(* CoDeSys 2.3 project: cy-221-wg-002.pro *)
(* Title: ClevergyAS - Albino E-02 *)
(* Version: 1.25 *)
(* Author: Andrea Ravasio *)
(* Libraries: mod_com.lib 2.12.10 13:48:32, SerComm.lib 31.5.11 07:54:36, Serial_Interface_01.lib 22.4.13 11:50:14, Standard.lib 2.12.10 13:48:34, SysLibTime.lib 2.12.10 13:48:32, Util.lib 26.9.14 09:12:46, Modb_l05.lib 13.5.15 09:30:08, Visual.lib 2.12.10 13:48:34, Ethernet.lib 2.12.10 13:48:32, WagoLibIdent.lib 25.2.13 10:12:16, WagoLibMBX_01.lib 20.3.12 15:32:40, WagoLibStatus.lib 2.12.10 13:48:32, SysLibFile.lib 2.12.10 13:48:34, SysLibRtc.lib 2.12.10 13:48:32, SysLibSockets.lib 10.2.11 08:20:54, SysLibEvent.lib 2.12.10 13:48:34, SysLibPlcCtrl.lib 2.12.10 13:48:32, SysLibCallback.lib 2.12.10 13:48:32, WagoLibModbus_IP_01.lib 24.7.13 14:05:58, WagoLibInfo.lib 25.2.13 09:58:44 *)

(* PLC configuration (modules and I/O channels)
0750-0402 4 DI 24 V DC 3.0ms [Type_1_4_Channels] node 0, in %IB0 out %QB0 {INTTypePAAssignment = PLC; INTTypeModule = plugged}
  AT %IX0.0 [BOOLOnX_I] Ch_1 Digital input
  AT %IX0.1 [BOOLOnX_I] Ch_2 Digital input
  AT %IX0.2 [BOOLOnX_I] Ch_3 Digital input
  AT %IX0.3 [BOOLOnX_I] Ch_4 Digital input
Fieldbus variables [FB_VARS] node 1, in %IB0 out %QB0
Flag variables [FLAG_VARS] node 2, in %IB0 out %QB0
Modbus-Master [MB_MASTER] node 3, in %IB0 out %QB0
*)

(* Global variable list: Addiitonal_Constants *)
VAR_GLOBAL CONSTANT

	Logger_MaxBCK : WORD:=100;

END_VAR

(* Global variable list: Additional_Retain *)
VAR_GLOBAL RETAIN PERSISTENT
	LogBCKIndex:  WORD;
END_VAR

(* Global variable list: Global_Constants *)
VAR_GLOBAL CONSTANT

	Plant_NAME		: STRING :='cySN:221  cyVER:0 - EGM Impianto Luci ';
	Plant_SN			: DWORD  :=221; 	         (* S/N Impianto di telecontrollo *)
	Plant_SW_VER		: WORD   :=0;		(* Versione SW installata *)


	(* Plant-dependent constants *)
	MAX_LUXNUM 								: INT :=12;
	MAX_LuxElement							: INT :=12;

	(* Filesystem *)
	FilesPath  			: STRING :='S:\';

	(* TCP Logger *)
	Logger_SERVER		: STRING:='';
	Logger_IP			: STRING:='178.33.227.41'; (*'192.168.100.3';*)
	Logger_PORT			: WORD  :=80;
	Logger_GETSTART		: STRING:='GET /cygmsrv/hsgm.ashx?';
	Logger_GETEND		: STRING:='$R$N$R$N';
	Logger_CHECK		: STRING:='True';
	Logger_CRLF			: STRING:='$R$N';
	Logger_DataFile		: STRING:='S:\LOG.DAT';
	Logger_DataFileOld	: STRING:='S:\LOG.BCK';
	Logger_IndexFile	: STRING:='S:\LOG.IDX';
	Logger_ConnRetries	: BYTE:=5;
	Logger_RecoverMsgs	: BYTE:=25;

	(* TCP Remote *)
	Remote_PORT			: WORD  :=10;
	Remote_WELCOME		: STRING:='Connected$R$N';
	Remote_OK			: STRING:='OK$R$N';
	Remote_ERROR		: STRING:='ERROR$R$N';

	(* TCP Sockets *)
	MAX_SEND_TCP_SERVER					 : DWORD:=60000;(*60000*)
	MAX_RECEIVE_TCP_SERVER				 : DWORD:=3000;
	MAX_RECEIVE_TCP_SERVER_SOCKET	 	 : DWORD:=3000;
	MAX_SEND_TCP_CLIENT					 : DWORD:=21000;(*15000*)
	MAX_RECEIVE_TCP_CLIENT				 : DWORD:=3000;
	MAX_RECEIVE_TCP_CLIENT_SOCKET		 : DWORD:=3000;
	MAX_RECEIVE_UDP_SERVER				 : INT  :=1472;
	MAX_RECEIVE_UDP_CLIENT				 : INT  :=1472;
	CONNECT_WATCHDOG_TIME				 : TIME :=t#10s;


	(* VISU COLORS *)
	COLOR_RED 			: DWORD:=16#2020F0;
	COLOR_YELLOW		: DWORD:=16#20F0F0;
	COLOR_GREEN			: DWORD:=16#20F020;
	COLOR_GREEN_OFF 	: DWORD:=16#006000;
	COLOR_LBLUE			: DWORD:=16#F0F080;
	COLOR_LIGHT_GREEN	: DWORD := 16#006000;


END_VAR

(* Global variable list: Global_Retain *)
VAR_GLOBAL RETAIN PERSISTENT

	Mode_Manual : BOOL := FALSE;

	WORKINGTIME_n : ARRAY[1..MAX_LUXNUM] OF DWORD;
	POWERONCYCLES_n : ARRAY[1..MAX_LUXNUM] OF WORD;
	ENERGYCOUNTER_n  : ARRAY[1..MAX_LUXNUM] OF WORD;
	ENERGYCOUNTER_T_n : ARRAY[1..MAX_LUXNUM] OF DWORD;

END_VAR

(* Global variable list: Global_Variables *)
VAR_GLOBAL

	SYS    : typ_SYS;
	Logger : typ_Logger;

	Lamp	:	LAMP_AL_GENERALE;
	LAMP_AL:BOOL; (* Dichiarata perchè non c'è l'uscita fisica *)
	T_AMB	:	INT;		(* Environment temperature *)

	(* Nodi Ethernet *)

	(* Analizzatori di rete Lovato DME 310 T2 *)
	ANZ01	:obj_Anz_Lovato_ETH := (ID:=1, IP:='192.168.2.84');		(* FONDERIA - CONTATORE N.1 *)
	ANZ02	:obj_Anz_Lovato_ETH := (ID:=2, IP:='192.168.2.85');		(* FONDERIA - CONTATORE N.2 *)
	ANZ03	:obj_Anz_Lovato_ETH := (ID:=3, IP:='192.168.2.86');		(* CAMPATA 1-2 - CONTATORE N.3*)
	ANZ04	:obj_Anz_Lovato_ETH := (ID:=4, IP:='192.168.2.87');		(* CAMPATA 3 - CONTATORE N.4 *)
	ANZ05	:obj_Anz_Lovato_ETH := (ID:=5, IP:='192.168.2.88');		(* CAMPATA 4 - CONTATORE N.5 *)
	ANZ06	:obj_Anz_Lovato_ETH := (ID:=6, IP:='192.168.2.89');		(* CAMPATA 5 - CONTATORE N.6 *)
	ANZ07	:obj_Anz_Lovato_ETH := (ID:=7, IP:='192.168.2.90');		(* CAMPATA 6 - CONTATORE N.7 *)
	ANZ08	:obj_Anz_Lovato_ETH := (ID:=8, IP:='192.168.2.91');		(* CAMPATA 7 - CONTATORE N.8 *)
	ANZ09	:obj_Anz_Lovato_ETH := (ID:=9, IP:='192.168.2.92');		(* CAMPATA 8 - CONTATORE N.9 *)
	ANZ10	:obj_Anz_Lovato_ETH := (ID:=10, IP:='192.168.2.93');		(* CAMPATA 9 - CONTATORE N.10 *)
	ANZ11	:obj_Anz_Lovato_ETH := (ID:=11, IP:='192.168.2.94');		(* MAGAZZINO - CONTATORE N.11 *)


	(* Nodi di rete I/ remoto SENECA ZE-4DI-2AI-2DO *)
	NODO01	:obj_Anz_Seneca_ETH := (ID:=1, IP:='192.168.2.95');		(* FONDERIA - CONTATORE N.1 e FONDERIA - CONTATORE N.2*)
	NODO02	:obj_Anz_Seneca_ETH := (ID:=2, IP:='192.168.2.96');		(* CAMPATA 1-2 - CONTATORE N.3 *)
	NODO03	:obj_Anz_Seneca_ETH := (ID:=3, IP:='192.168.2.97');		(* CAMPATA 3 - CONTATORE N.4 *)
	NODO04	:obj_Anz_Seneca_ETH := (ID:=4, IP:='192.168.2.98');		(* CAMPATA 4 - CONTATORE N.5 *)
	NODO05	:obj_Anz_Seneca_ETH := (ID:=5, IP:='192.168.2.99');		(* CAMPATA 5 - CONTATORE N.6 *)
	NODO06	:obj_Anz_Seneca_ETH := (ID:=6, IP:='192.168.2.103');		(* CAMPATA 6 - CONTATORE N.7 *)
	NODO07	:obj_Anz_Seneca_ETH := (ID:=7, IP:='192.168.2.104');		(* CAMPATA 7 - CONTATORE N.8 *)
	NODO08	:obj_Anz_Seneca_ETH := (ID:=8, IP:='192.168.2.105');		(* CAMPATA 8 - CONTATORE N.9 *)
	NODO09	:obj_Anz_Seneca_ETH := (ID:=9, IP:='192.168.2.107');		(* CAMPATA 9 - CONTATORE N.10 *)
	NODO10	:obj_Anz_Seneca_ETH := (ID:=10, IP:='192.168.2.106');	(* MAGAZZINO - CONTATORE N.11 *)

(*	LuxElement : ARRAY[1..MAX_LuxElement] OF obj_LUX:=( dimmingtype:=0, CTRL_MODE:=2,CTRL_MODE_BackUp:=2, KeyQty:=1, KeyMode:=SWITCH_NO);
	TabDefaultLux : ARRAY[1..MAX_LuxElement] OF type_TabListLux :=(LuxNumber:=1, Mode:=2) ; *)
 
	LuxElement01: 	obj_LuxSimple:=( ID:=1,CTRL_MODE:=2);
	LuxElement02: 	obj_LuxSimple:=( ID:=2,CTRL_MODE:=2);
	LuxElement03: 	obj_LuxSimple:=( ID:=3, CTRL_MODE:=2);
	LuxElement04: 	obj_LuxSimple:=( ID:=4, CTRL_MODE:=2);
	LuxElement05: 	obj_LuxSimple:=( ID:=5, CTRL_MODE:=2);
	LuxElement06: 	obj_LuxSimple:=( ID:=6, CTRL_MODE:=2);
	LuxElement07: 	obj_LuxSimple:=( ID:=7, CTRL_MODE:=2);
	LuxElement08: 	obj_LuxSimple:=( ID:=8, CTRL_MODE:=2);
	LuxElement09: 	obj_LuxSimple:=( ID:=9, CTRL_MODE:=2);
	LuxElement10: 	obj_LuxSimple:=( ID:=10, CTRL_MODE:=2);
	LuxElement11: 	obj_LuxSimple:=( ID:=11, CTRL_MODE:=2);
	LuxElement12: 	obj_LuxSimple:=( ID:=12, CTRL_MODE:=2);


	(* Crono per gestione accensioni luci impostazione lux *)
	CRON01	:	obj_CRONTER_01 := (ID:=1, Local_MaxRunTAmb:=5000,Histeresys:=50,TipoCrono:='CRONG'(* Riferimento nle file LOG *));
	CRON02	:	obj_CRONTER_01 := (ID:=2, Local_MaxRunTAmb:=5000,Histeresys:=50,TipoCrono:='CRONG'(* Riferimento nle file LOG *));
	CRON03	:	obj_CRONTER_01 := (ID:=3, Local_MaxRunTAmb:=5000,Histeresys:=50,TipoCrono:='CRONG'(* Riferimento nle file LOG *));
	CRON04	:	obj_CRONTER_01:=  (ID:=4, Local_MaxRunTAmb:=5000,Histeresys:=50,TipoCrono:='CRONG'(* Riferimento nle file LOG *));
	CRON05	:	obj_CRONTER_01 := (ID:=5, Local_MaxRunTAmb:=5000,Histeresys:=50,TipoCrono:='CRONG'(* Riferimento nle file LOG *));
	CRON06	:	obj_CRONTER_01 := (ID:=6, Local_MaxRunTAmb:=5000,Histeresys:=50,TipoCrono:='CRONG'(* Riferimento nle file LOG *));
	CRON07	:	obj_CRONTER_01 := (ID:=7, Local_MaxRunTAmb:=5000,Histeresys:=50,TipoCrono:='CRONG'(* Riferimento nle file LOG *));
	CRON08	:	obj_CRONTER_01 := (ID:=8, Local_MaxRunTAmb:=5000,Histeresys:=50,TipoCrono:='CRONG'(* Riferimento nle file LOG *));
	CRON09	:	obj_CRONTER_01 := (ID:=9, Local_MaxRunTAmb:=5000,Histeresys:=50,TipoCrono:='CRONG'(* Riferimento nle file LOG *));
	CRON10	:	obj_CRONTER_01 := (ID:=10, Local_MaxRunTAmb:=5000,Histeresys:=50,TipoCrono:='CRONG'(* Riferimento nle file LOG *));
	CRON11	:	obj_CRONTER_01 := (ID:=11, Local_MaxRunTAmb:=5000,Histeresys:=50,TipoCrono:='CRONG'(* Riferimento nle file LOG *));
	CronEd	: 	obj_CRON_EDITOR_01;






	KEYON :BOOL;




(* CONFIGURAZIONE INGRESSI ANALOGICI 4-20mA per oggetti ZTHL  *)

	(* FONDERIA - CONTATORE N.1 e FONDERIA - CONTATORE N.2*)
	ZTHL01  : obj_AI_GEN	:= ( ID:=1 ,
								SogliaHL:=3000 ,   	 	(* Soglia Sonda Aperta = 2,5mA *)
								SogliaHH:=20500,	 	(* Soglia Sonda CC = 20mA *)
								SogliaWL:=-100, 			(* Soglia WRN Bassa  *)
								SogliaWH:=1020,			(* Soglia WRN Alta   *)
								PuntoMinX:=0, 		   	(* Scalatura Minima vedi data di targa sonda 0 LUX *)
								PuntoMaxX:=1000,		(* Scalatura Massima Vedi data di targa Sonda  500 LUXr *)
								PuntoMinY:=4000,		(* Valore minimio per scalatura = 4mA *)
								PuntoMaxY:=20000,		(* Valore Massimo per Scalatura = 20mA *)
								Decimali:=0,			(* Decimali da ottenere durante la scalatura *)
								TipoSensore:='LUXMETER'		(* Riferimento nle file LOG *)
								);

	(* CAMPATA 1-2 - CONTATORE N.3 *)
	ZTHL02  : obj_AI_GEN	:= ( ID:=2 ,
								SogliaHL:=3000 ,   	 	(* Soglia Sonda Aperta = 2,5mA *)
								SogliaHH:=20500,	 	(* Soglia Sonda CC = 20mA *)
								SogliaWL:=-100, 			(* Soglia WRN Bassa  *)
								SogliaWH:=1020,			(* Soglia WRN Alta   *)
								PuntoMinX:=0, 		   	(* Scalatura Minima vedi data di targa sonda 0 LUX *)
								PuntoMaxX:=1000,		(* Scalatura Massima Vedi data di targa Sonda  500 LUXr *)
								PuntoMinY:=4000,		(* Valore minimio per scalatura = 4mA *)
								PuntoMaxY:=20000,		(* Valore Massimo per Scalatura = 20mA *)
								Decimali:=0,			(* Decimali da ottenere durante la scalatura *)
								TipoSensore:='LUXMETER'		(* Riferimento nle file LOG *)								);
	(* CAMPATA 3 - CONTATORE N.4 *)
	ZTHL03  : obj_AI_GEN	:= ( ID:=3 ,
								SogliaHL:=3000 ,   	 	(* Soglia Sonda Aperta = 2,5mA *)
								SogliaHH:=20500,	 	(* Soglia Sonda CC = 20mA *)
								SogliaWL:=-100, 			(* Soglia WRN Bassa  *)
								SogliaWH:=1020,			(* Soglia WRN Alta   *)
								PuntoMinX:=0, 		   	(* Scalatura Minima vedi data di targa sonda 0 LUX *)
								PuntoMaxX:=1000,		(* Scalatura Massima Vedi data di targa Sonda  500 LUXr *)
								PuntoMinY:=4000,		(* Valore minimio per scalatura = 4mA *)
								PuntoMaxY:=20000,		(* Valore Massimo per Scalatura = 20mA *)
								Decimali:=0,			(* Decimali da ottenere durante la scalatura *)
								TipoSensore:='LUXMETER'		(* Riferimento nle file LOG *)
								);
	(* CAMPATA 4 - CONTATORE N.5 *)
	ZTHL04  : obj_AI_GEN	:= ( ID:=4 ,
								SogliaHL:=3000 ,   	 	(* Soglia Sonda Aperta = 2,5mA *)
								SogliaHH:=20500,	 	(* Soglia Sonda CC = 20mA *)
								SogliaWL:=-100, 			(* Soglia WRN Bassa  *)
								SogliaWH:=1020,			(* Soglia WRN Alta   *)
								PuntoMinX:=0, 		   	(* Scalatura Minima vedi data di targa sonda 0 LUX *)
								PuntoMaxX:=1000,		(* Scalatura Massima Vedi data di targa Sonda  500 LUXr *)
								PuntoMinY:=4000,		(* Valore minimio per scalatura = 4mA *)
								PuntoMaxY:=20000,		(* Valore Massimo per Scalatura = 20mA *)
								Decimali:=0,			(* Decimali da ottenere durante la scalatura *)
								TipoSensore:='LUXMETER'		(* Riferimento nle file LOG *)
								);
	(* CAMPATA 5 - CONTATORE N.6 *)
	ZTHL05  : obj_AI_GEN	:= ( ID:=5 ,
								SogliaHL:=3000 ,   	 	(* Soglia Sonda Aperta = 2,5mA *)
								SogliaHH:=20500,	 	(* Soglia Sonda CC = 20mA *)
								SogliaWL:=-100, 			(* Soglia WRN Bassa  *)
								SogliaWH:=1020,			(* Soglia WRN Alta   *)
								PuntoMinX:=0, 		   	(* Scalatura Minima vedi data di targa sonda 0 LUX *)
								PuntoMaxX:=1000,		(* Scalatura Massima Vedi data di targa Sonda  500 LUXr *)
								PuntoMinY:=4000,		(* Valore minimio per scalatura = 4mA *)
								PuntoMaxY:=20000,		(* Valore Massimo per Scalatura = 20mA *)
								Decimali:=0,			(* Decimali da ottenere durante la scalatura *)
								TipoSensore:='LUXMETER'		(* Riferimento nle file LOG *)
								);
	(* CAMPATA 6 - CONTATORE N.7 *)
	ZTHL06  : obj_AI_GEN	:= ( ID:=6 ,
								SogliaHL:=3000 ,   	 	(* Soglia Sonda Aperta = 2,5mA *)
								SogliaHH:=20500,	 	(* Soglia Sonda CC = 20mA *)
								SogliaWL:=-100, 			(* Soglia WRN Bassa  *)
								SogliaWH:=1020,			(* Soglia WRN Alta   *)
								PuntoMinX:=0, 		   	(* Scalatura Minima vedi data di targa sonda 0 LUX *)
								PuntoMaxX:=1000,		(* Scalatura Massima Vedi data di targa Sonda  500 LUXr *)
								PuntoMinY:=4000,		(* Valore minimio per scalatura = 4mA *)
								PuntoMaxY:=20000,		(* Valore Massimo per Scalatura = 20mA *)
								Decimali:=0,			(* Decimali da ottenere durante la scalatura *)
								TipoSensore:='LUXMETER'		(* Riferimento nle file LOG *)
								);
	(* CAMPATA 7 - CONTATORE N.8 *)
	ZTHL07  : obj_AI_GEN	:= ( ID:=7 ,
								SogliaHL:=3000 ,   	 	(* Soglia Sonda Aperta = 2,5mA *)
								SogliaHH:=20500,	 	(* Soglia Sonda CC = 20mA *)
								SogliaWL:=-100, 			(* Soglia WRN Bassa  *)
								SogliaWH:=1020,			(* Soglia WRN Alta   *)
								PuntoMinX:=0, 		   	(* Scalatura Minima vedi data di targa sonda 0 LUX *)
								PuntoMaxX:=1000,		(* Scalatura Massima Vedi data di targa Sonda  500 LUXr *)
								PuntoMinY:=4000,		(* Valore minimio per scalatura = 4mA *)
								PuntoMaxY:=20000,		(* Valore Massimo per Scalatura = 20mA *)
								Decimali:=0,			(* Decimali da ottenere durante la scalatura *)
								TipoSensore:='LUXMETER'		(* Riferimento nle file LOG *)
								);
	(* CAMPATA 8 - CONTATORE N.9 *)
	ZTHL08  : obj_AI_GEN	:= ( ID:=8 ,
								SogliaHL:=3000 ,   	 	(* Soglia Sonda Aperta = 2,5mA *)
								SogliaHH:=20500,	 	(* Soglia Sonda CC = 20mA *)
								SogliaWL:=-100, 			(* Soglia WRN Bassa  *)
								SogliaWH:=1020,			(* Soglia WRN Alta   *)
								PuntoMinX:=0, 		   	(* Scalatura Minima vedi data di targa sonda 0 LUX *)
								PuntoMaxX:=1000,		(* Scalatura Massima Vedi data di targa Sonda  500 LUXr *)
								PuntoMinY:=4000,		(* Valore minimio per scalatura = 4mA *)
								PuntoMaxY:=20000,		(* Valore Massimo per Scalatura = 20mA *)
								Decimali:=0,			(* Decimali da ottenere durante la scalatura *)
								TipoSensore:='LUXMETER'		(* Riferimento nle file LOG *)
								);
	(* CAMPATA 9 - CONTATORE N.10 *)
	ZTHL09  : obj_AI_GEN	:= ( ID:=9 ,
								SogliaHL:=3000 ,   	 	(* Soglia Sonda Aperta = 2,5mA *)
								SogliaHH:=20500,	 	(* Soglia Sonda CC = 20mA *)
								SogliaWL:=-100, 			(* Soglia WRN Bassa  *)
								SogliaWH:=1020,			(* Soglia WRN Alta   *)
								PuntoMinX:=0, 		   	(* Scalatura Minima vedi data di targa sonda 0 LUX *)
								PuntoMaxX:=1000,		(* Scalatura Massima Vedi data di targa Sonda  500 LUXr *)
								PuntoMinY:=4000,		(* Valore minimio per scalatura = 4mA *)
								PuntoMaxY:=20000,		(* Valore Massimo per Scalatura = 20mA *)
								Decimali:=0,			(* Decimali da ottenere durante la scalatura *)
								TipoSensore:='LUXMETER'		(* Riferimento nle file LOG *)
								);
	(* MAGAZZINO - CONTATORE N.11 *)
	ZTHL10  : obj_AI_GEN	:= ( ID:=10 ,
								SogliaHL:=3000 ,   	 	(* Soglia Sonda Aperta = 2,5mA *)
								SogliaHH:=20500,	 	(* Soglia Sonda CC = 20mA *)
								SogliaWL:=-100, 			(* Soglia WRN Bassa  *)
								SogliaWH:=1020,			(* Soglia WRN Alta   *)
								PuntoMinX:=0, 		   	(* Scalatura Minima vedi data di targa sonda 0 LUX *)
								PuntoMaxX:=1000,		(* Scalatura Massima Vedi data di targa Sonda  500 LUXr *)
								PuntoMinY:=4000,		(* Valore minimio per scalatura = 4mA *)
								PuntoMaxY:=20000,		(* Valore Massimo per Scalatura = 20mA *)
								Decimali:=0,			(* Decimali da ottenere durante la scalatura *)
								TipoSensore:='LUXMETER'		(* Riferimento nle file LOG *)
								);







END_VAR

(* Data type in Errors *)
TYPE en_Logger_ErrLev :
(
	EL_Log			:=0,
	EL_Wrn			:=1,
	EL_Alarm		:=2,
	EL_AlarmStop	:=3
);
END_TYPE

(* Data type in Errors *)
TYPE en_Logger_Status :
(
	S_Logger_UNKNOWN := 0,
	S_Logger_IDLE,
	S_Logger_WAITCONN,
	S_Logger_WAITTX,
	S_Logger_WAITRESP,
	S_Logger_ERROR
);
END_TYPE

(* Data type *)
TYPE en_Modbus_Reg_Type :
(
	VALUE_REAL		:=0,
	VALUE_LONG		:=4
);
END_TYPE

(* Data type *)
TYPE en_SYS_Objects :
(
	EO_SYS		:=0,  (* PLC *)
	EO_VPN		:=1,  (* VPN *)
	EO_DOOR		:=2,  (* Door & access control *)

	EO_CAL		:=10, (* Caldaia *)
	EO_CIR		:=11, (* Circolatore *)
	EO_CRON		:=12, (* Crono-termostato *)
	EO_VRD		:=13, (* Valvola miscelatore pannelli *)
	EO_CTL		:=14, (* Contalitri *)
	EO_CTB		:=15, (* Contabilizzatore *)
	EO_TPV		:=16, (* Temperature probes values *)
	EO_PPV		:=17, (* Pressure probes values *)
	EO_PBV		:=18, (* Over-Pressure Alarms *)
	EO_TBV		:=19, (* Over-Temperature Alarms *)
	EO_PMV		:=20, (* Under-Pressure Alarms *)
	EO_GRU		:=21, (* Gruppo termico *)
	EO_PDC		:=22, (* Pompa di calore *)
	EO_SOL		:=23, (* Pannello solare termico *)
	EO_ESOL		:=24, (* Pannello solare fotovoltaico *)
	EO_GAS		:=25, (* Contatore GAS *)
	EO_PORT		:=26, (* Misuratore di portata *)
	EO_FPV		:=27, (* Flow probes values *)
	EO_ANZ		:=28, (* Analizzatore di rete *)
	EO_SCA		:=29, (* Signal Control Alarms *)
	EO_LUX		:=30, (* Base Illumination point *)
	EO_LUXM		:=31, (* Metered Illumination point *)
	EO_PSG		:=32, (* Sensore di passaggio *)
	EO_HVAC		:=33, (* Heating, Ventilating and Air Conditioning *)
	EO_HYGRV	:=34, (* Relative Humidity sensors value *)
	EO_COOV		:=35, (* Carbon Dioxide CO2 sensors value *)
	EO_INV			:=36, (* Inverter *)
	EO_STR		:=37, (* Smart string box *)

	EO_CIRD		:=39, (* Double CIR *)
	EO_ACS		:=40, (* Hot domestic water *)
	EO_FRG		:=41, (* Frigo *)
	EO_THER		:=42, (* Thermostat *)
	EO_CIRM		:=43, (* Modbus CIR *)
	EO_CIRDM	:=44, (* Modbus double CIR *)
	EO_UTA		:=47, (* Modbus double CIR *)

	EO_FPT		:=53, (* Flow Pressure Temperature	FPTxx *)


	EO_ZGW			:=200,  (* ZigBee - Gateway *)
	EO_ZRM			:=201,	(* ZigBee - Repeater *)
	EO_ZREL			:=202,	(* ZigBee - Actuator rele *)
	EO_ZTHL			:=203,	(* ZigBee - Temperature Sensor *)

	EO_ASGW			:=250,	(* ASi - Gateway *)
	EO_ASCBI		:=251,	(* ASi - Input Board, Ciabatta *)

	EO_LON			:=1000, (* Bus - LON *)
	EO_MODBUS		:=1001, (* Bus - MODBUS *)
	EO_MBUS			:=1002, (* Bus - M-BUS *)
	EO_MODBUS_TCP	:=1003, (* Bus - MODBUS TCP *)

	EO_VAR 			:=3000, (* Variabili Generali di Set e Get *)


	EO_COMPINGRR		:=10000,		(*Compressore Ingerson Rand R225 NE *)
	EO_COMPINGRML	:=	10001,		(*Compressore Ingerson Rand ML250SSR *)
	EO_ESC				:=	10002,		(*Essicatore *)





	EO_GENERIC		:=9000, (* Generic dataset *)
	EO_EXPO			:=9001 (* EXPO dataset *)
);
END_TYPE

(* Data type *)
TYPE en_SYS_Status :
(
	S_UNKNOWN  := 0,
	S_STARTUP,
	S_INIT_RTC,
	S_INIT_VAR,
	S_AUTOTEST,
	S_RUNNING,
	S_SHUTDOWN,
	S_HALT
);
END_TYPE

(* Data type *)
(*
	typ_ANZ_3P 

	Data that each ANZ 3-phase block must provide (to the Clevergy platform).
*)
TYPE typ_ANZ_REAL :
STRUCT

	(* voltages *)
	V_L1N		:	REAL;	(* V *)
	V_L2N		:	REAL;
	V_L3N		:	REAL;
	V_L1L2		:	REAL;
	V_L2L3		:	REAL;
	V_L3L1		:	REAL;

	(* frequency *)
	FREQ		:	REAL;	(* E-3 Hz *) (* rif. L1 *)

	(* currents *)
	I_L1			:	REAL;	(* E-3 A *)
	I_L2			:	REAL;
	I_L3			:	REAL;
	I_L1_Max		:	REAL;	(* E-3 A *)
	I_L2_Max		:	REAL;
	I_L3_Max		:	REAL;

	(* power factors *)
	PF_L1		:	REAL;	(* E-3 *)
	PF_L2		:	REAL;
	PF_L3		:	REAL;

	(* active powers *)
	P_3P			:	REAL;   (* W *)
	P_3P_Avg		:	REAL;
	P_3P_Max	:	REAL:=0;

	(* reactive powers *)
	Q_3P		:	REAL;	(* VAr *)
	Q_3P_Max	:	REAL:=-2147483648;	(* VAr *)

	(* active energy *)
	WH_3P		:	REAL;	(* Wh *)

	(* reactive energy *)
	VARH_3P		:	REAL;	(* VArh *)

	(* cosphi *)
	COSPHI_L1		:	REAL;	(* E-3 *)
	COSPHI_L2		:	REAL;	(* E-3 *)
	COSPHI_L3		:	REAL;	(* E-3 *)

END_STRUCT
END_TYPE

(* Data type in Plant_Objects *)
TYPE typ_Clima : (* CURVA CLIMATICA *)
STRUCT
	InitOK:		BOOL;
	Points: 	ARRAY [0..10] OF POINT;
END_STRUCT
END_TYPE

(* Data type in Plant_Objects *)
TYPE typ_Cron_Calendar :
STRUCT
	Profile		: ARRAY[0..384] OF BYTE;
END_STRUCT
END_TYPE

(* Data type in Plant_Objects *)
TYPE typ_Cron_Jolly :
STRUCT
	Start		: DT;
	End			: DT;
	Temp		: WORD;
	Flags		: WORD; (* B0:Enabled B1..B15:Unused *)
END_STRUCT
END_TYPE

(* Data type in Plant_Objects *)
TYPE typ_Cron_Profile :
STRUCT
	Flags		: WORD;
	Setpoint	: ARRAY [0..95] OF WORD;
END_STRUCT
END_TYPE

(* Data type in Errors *)
TYPE typ_Logger :
STRUCT
	Status		: en_Logger_Status;

	SendReq		: BOOL;
	SendIdx		: DWORD;
	SendData	: ARRAY [0..MAX_SEND_TCP_CLIENT] OF BYTE;
	SendLen		: DINT;

	TData		: ARRAY [0..MAX_SEND_TCP_CLIENT] OF BYTE;
	TLen		: DINT;

	LastIdxPos	: DWORD;

	(* Temporary variables used by objects *)
	s1			: STRING(256);
	i1			: WORD;


END_STRUCT
END_TYPE

(* Data type in Plant_Objects *)
TYPE typ_MODBUS_VAR : (* Gestione parametri MODBUS *)
STRUCT
	SlaveAddress	: BYTE;
	FunCode			: BYTE;
	FunAddress		: WORD;
	Refresh_Time	: BYTE; (* 0:No refresh x:Refresh in seconds *)
	Refresh_Cnt		: BYTE; (* INTERNAL *)
	Variable		: POINTER TO WORD;
	Variable_Size	: BYTE;
	Variable_Mirror : WORD; (* INTERNAL [Force refresh on read variables when <>0] *)
END_STRUCT
END_TYPE

(* Data type in Plant_Objects *)
TYPE typ_MODBUS_VAR_ANZ : (* Gestione parametri MODBUS *)
STRUCT
	SlaveAddress	: BYTE;
	FunCode			: BYTE;
	FunAddress		: WORD;
	Refresh_Time	: BYTE; (* 0:No refresh x:Refresh in seconds *)
	Refresh_Cnt		: BYTE; (* INTERNAL *)
	Variable		: POINTER TO ARRAY [0..124] OF WORD;	(* For classical ModBus it has to be equal to "typModbusResponse.Data"
																that is an array of 125 word ([0..124]) *)
	Variable_Size	: BYTE;
	Variable_Mirror : WORD; (* INTERNAL [Force refresh on read variables when <>0] *)
END_STRUCT
END_TYPE

(* Data type *)
TYPE typ_SYS :
STRUCT
	Status			: en_SYS_Status;
	Warning			: BOOL;
	Alarm			: BOOL;
	AlarmStop		: BOOL;

	Time_LogString	: STRING;
	Time_Year		: WORD;
	Time_Month		: BYTE;
	Time_Day		: BYTE;

	Time_CT_DT		: DT;
	Time_CT_Day		: WORD;
	Time_CT_Quarter	: BYTE;

	LastLogs_Idx	: BYTE;
	LastLogs_Dat	: ARRAY[0..5] OF STRING;
	LastLogs_Msg	: ARRAY[0..5] OF STRING;

END_STRUCT
END_TYPE

(* POU PLC_PRG, ST *)
PROGRAM PLC_PRG
VAR
	Timer1: TON; (* Fast controls tick *)
	Timer2: TON; (* Plant control tick *)
	Timer3: TON; (* Logger timer *)


	status : BYTE;
	i	  : BYTE;
	loggando:BOOL:=FALSE;

	HMI_AggiornaLog: BOOL;


	EseguiLog: INT;
	Ton_pausaTrig: TON;
	R_TrigAggiornaLog: R_TRIG;


	TempoLog: TIME := t#1s;
	Pippo1: STRING;
	Pippo2: STRING;




	IndiceAnz: INT;
	typeVisuANZ :typ_ANZ_real;
	VisuTestoANZ: ARRAY [1..2,1..26] OF STRING;
	BitStart01: BOOL;
	BitStart02: BOOL;
	BitStart03: BOOL;
	BitStart04: BOOL;
	BitStart05: BOOL;
	BitStart06: BOOL;
	BitStart07: BOOL;
	BitStart08: BOOL;
	BitStart09: BOOL;
	BitStart10: BOOL;
	BitStart11: BOOL;
	BitStart12: BOOL;


END_VAR

VAR_INPUT RETAIN
	(* gestione lux *)
	SogliaLux01:INT:=250;
	IsteresiLux01:INT:=100;
	SogliaLux02:INT:=400;
	IsteresiLux02:INT:=20;
	SogliaLux03:INT:=450;
	IsteresiLux03:INT:=20;
	SogliaLux04:INT:=400;
	IsteresiLux04:INT:=20;
	SogliaLux05:INT:=480;
	IsteresiLux05:INT:=20;
	SogliaLux06:INT:=480;
	IsteresiLux06:INT:=20;
	SogliaLux07:INT:=350;
	IsteresiLux07:INT:=20;
	SogliaLux08:INT:=400;
	IsteresiLux08:INT:=20;
	SogliaLux09:INT:=490;
	IsteresiLux09:INT:=20;
	SogliaLux10:INT:=480;
	IsteresiLux10:INT:=20;
	SogliaLux11:INT:=400;
	IsteresiLux11:INT:=20;
	SogliaLux12:INT:=450;
	IsteresiLux12:INT:=20;
	delayOffLux:INT:=300;

	ToffDelayLux1 : TOF;
	ToffDelayLux2 : TOF;
	ToffDelayLux3 : TOF;
	ToffDelayLux4 : TOF;
	ToffDelayLux5 : TOF;
	ToffDelayLux6 : TOF;
	ToffDelayLux7 : TOF;
	ToffDelayLux8 : TOF;
	ToffDelayLux9 : TOF;
	ToffDelayLux10 : TOF;
	ToffDelayLux11 : TOF;
	ToffDelayLux12 : TOF;





END_VAR

VAR_INPUT
	RichiestaDaRemoto:BOOL;

END_VAR
(******************************************************************************
 ****                           MAIN TASK CODE                             ****
 ******************************************************************************

	Network setup:
		IP  = 192.168.2.73 | MSK = 255.255.255.0
		GW	= 192.168.2.254 | DNS = 192.168.100.1
		SNTP = 193.204.114.232 (3600s) ==> 192.168.100.3
*)






(*==============================*)
(*===== Main status machine ====*)
(*==============================*)


Main_Stm();

(*==============================*)
(*== Running cycle operations ==*)
(*==============================*)

IF SYS.Status>S_INIT_VAR THEN

 	ANZ01();
	ANZ02();
	ANZ03();
	ANZ04();
	ANZ05();
	ANZ06();
	ANZ07();
	ANZ08();
	ANZ09();
	ANZ10();
	ANZ11();


	NODO01();
	NODO02();
	NODO03();
	NODO04();
	NODO05();
	NODO06();
	NODO07();
	NODO08();
	NODO09();
	NODO10();


(* limito le variabili di soglia Massima *)

	SogliaLux01:=LIMIT(0,SogliaLux01,ZTHL01.PuntoMaxX-1);
	SogliaLux02:=LIMIT(0,SogliaLux02,ZTHL02.PuntoMaxX-1);
	SogliaLux03:=LIMIT(0,SogliaLux03,ZTHL03.PuntoMaxX-1);
	SogliaLux04:=LIMIT(0,SogliaLux04,ZTHL04.PuntoMaxX-1);
	SogliaLux05:=LIMIT(0,SogliaLux05,ZTHL05.PuntoMaxX-1);
	SogliaLux06:=LIMIT(0,SogliaLux06,ZTHL06.PuntoMaxX-1);
	SogliaLux07:=LIMIT(0,SogliaLux07,ZTHL07.PuntoMaxX-1);
	SogliaLux08:=LIMIT(0,SogliaLux08,ZTHL08.PuntoMaxX-1);
	SogliaLux09:=LIMIT(0,SogliaLux09,ZTHL09.PuntoMaxX-1);
	SogliaLux10:=LIMIT(0,SogliaLux10,ZTHL10.PuntoMaxX-1);
	SogliaLux11:=LIMIT(0,SogliaLux11,ZTHL02.PuntoMaxX-1);
	SogliaLux12:=LIMIT(0,SogliaLux12,ZTHL03.PuntoMaxX-1);



END_IF


(*==============================*)
(*== System cycle operations ===*)
(*==============================*)
(* Execute TCP processes *)
Logger_Proc();
Remote_Proc();
(*
(* Update user led *)
USRLED_Update();*)

(* Execute Cron Editor commands *)
CronEd();
END_PROGRAM
ACTION Main_Stm:
CASE Sys.Status OF

	S_STARTUP:
		Sys.Status:=S_INIT_RTC;

	S_INIT_RTC:
		(* Check RTC and update from network *)
		RTC_Update();
		(* Check time *)
		IF Sys.Time_Year>2000 THEN
			Sys.Status:=S_INIT_VAR;
		END_IF








	S_INIT_VAR:
		LogEv(EL_Wrn,EO_SYS,0,1,CONCAT('System_startup_v',WORD_TO_STRING(Plant_SW_VER)));
		Sys.Status:=S_RUNNING;

	S_RUNNING:


		Timer1(IN:=NOT Timer1.Q,PT:=T#50ms);
		IF Timer1.Q THEN
			(* Update system checks *)
			SYS_Proc();
		END_IF




		Timer2(IN:=NOT Timer2.Q,PT:=T#500ms);
		IF Timer2.Q THEN


			(* Read current date/time *)
			RTC_Update();

			(* richiamo i crono *)    (* 1- FONDERIA - CONTATORE N.1-2
									2 - CAMPATA 1-2 - CONTATORE N.3
									3 - CAMPATA 3 - CONTATORE N.4
									4 - CAMPATA 4 - CONTATORE N.5
									5 - CAMPATA 5 - CONTATORE N.6
									6 - CAMPATA 6 - CONTATORE N.7
									7 - CAMPATA 7 - CONTATORE N.8
									8 - CAMPATA 8 - CONTATORE N.9
									9 - CAMPATA 9 - CONTATORE N.10
									10 - MAGAZZINO - CONTATORE N.11 *)
			CRON01();
			CRON02();
			CRON03();
			CRON04();
			CRON05();
			CRON06();
			CRON07();
			CRON08();
			CRON09();
			CRON10();





		(* Letttura ingressi analogici  *)

			ZTHL01	 ( AI_INPUT:=NODO01.AI_01 );
			ZTHL02	 ( AI_INPUT:=NODO02.AI_01 );
			ZTHL03	 ( AI_INPUT:=NODO03.AI_01 );
			ZTHL04	 ( AI_INPUT:=NODO04.AI_01 );
			ZTHL05	 ( AI_INPUT:=NODO05.AI_01 );
			ZTHL06	 ( AI_INPUT:=NODO06.AI_01 );
			ZTHL07	 ( AI_INPUT:=NODO07.AI_01 );
			ZTHL08	 ( AI_INPUT:=NODO08.AI_01 );
			ZTHL09	 ( AI_INPUT:=NODO09.AI_01 );
			ZTHL10	 ( AI_INPUT:=NODO10.AI_01 );



(*		LuxElement[1](ValInCronoInLux:=SEL(ASTR01.setPoint>0,0,1000),
						WORKINGTIME:=WORKINGTIME_n[1],
						POWERONCYCLES:=POWERONCYCLES_n[1],
						ENERGYCOUNTER:=ENERGYCOUNTER_n[1],
						ENERGYCOUNTER_t :=ENERGYCOUNTER_T_n[1],
						Lux_Enable => NODO01.w_DO_01,
						Lux_State:=(ANZ01.measures.P_3P>=LUXLEARN01.refValue));   *)







			(* FONDERIA - CONTATORE N.1 FONDERIA - CONTATORE N.2 *)

		IF   ZTHL01.ERR (*OR NODO01.Status_Log>0*) THEN
			BitStart01:=TRUE;
		ELSE
			IF ZTHL01.ValoreScalato <  SogliaLux01  THEN
				BitStart01:=TRUE;
			ELSIF   ZTHL01.ValoreScalato >   (LIMIT(0,SogliaLux01 + IsteresiLux01,ZTHL01.PuntoMaxX)) THEN
				BitStart01:=FALSE;
			END_IF;
		END_IF;
		ToffDelayLux1(IN:=BitStart01 AND CRON01.RunCrono, PT:= t#1s*delayOffLux, Q=> , ET=> );
		LuxElement01(DI_ONLux:=ToffDelayLux1.Q,
						Lux_State:=NODO01.DI_04,
						WORKINGTIME:=WORKINGTIME_n[1],
						POWERONCYCLES:=POWERONCYCLES_n[1],
						ENERGYCOUNTER:=ENERGYCOUNTER_n[1],
						ENERGYCOUNTER_t :=ENERGYCOUNTER_T_n[1],
						Lux_Enable => NODO01.w_DO_01,
						Lux_Auto:=NODO01.DI_01,
						Lux_Off:= NODO01.DI_02,
						Lux_Man:= NODO01.DI_03
						);

			(* CAMPATA 1-2 - CONTATORE N.3 *)

		IF   ZTHL02.ERR (*OR NODO02.Status_Log>0*) THEN
			BitStart02:=TRUE;
		ELSE
			IF ZTHL02.ValoreScalato <  SogliaLux02  THEN
				BitStart02:=TRUE;
			ELSIF   ZTHL02.ValoreScalato >  (LIMIT(0,SogliaLux02 + IsteresiLux02,ZTHL02.PuntoMaxX)) THEN
				BitStart02:=FALSE;
			END_IF;
		END_IF;
		ToffDelayLux2(IN:=BitStart02 AND CRON02.RunCrono, PT:= t#1s*delayOffLux, Q=> , ET=> );
		LuxElement02(DI_ONLux:=ToffDelayLux2.Q,
						Lux_State:=NODO02.DI_04,
						WORKINGTIME:=WORKINGTIME_n[1],
						POWERONCYCLES:=POWERONCYCLES_n[1],
						ENERGYCOUNTER:=ENERGYCOUNTER_n[1],
						ENERGYCOUNTER_t :=ENERGYCOUNTER_T_n[1],
						Lux_Enable => NODO02.w_DO_01,
						Lux_Auto:=NODO02.DI_01,
						Lux_Off:= NODO02.DI_02,
						Lux_Man:= NODO02.DI_03);

			(* CAMPATA 3 - CONTATORE N.4 *)

		IF   ZTHL03.ERR (*OR NODO03.Status_Log>0*) THEN
			BitStart03:=TRUE;
		ELSE
			IF ZTHL03.ValoreScalato <  SogliaLux03  THEN
				BitStart03:=TRUE;
			ELSIF   ZTHL03.ValoreScalato >   (LIMIT(0,SogliaLux03 + IsteresiLux03,ZTHL03.PuntoMaxX)) THEN
				BitStart03:=FALSE;
			END_IF;
		END_IF;
		ToffDelayLux3(IN:=BitStart03 AND CRON03.RunCrono, PT:= t#1s*delayOffLux, Q=> , ET=> );
		LuxElement03(DI_ONLux:=ToffDelayLux3.Q,
						Lux_State:=NODO03.DI_04,
						WORKINGTIME:=WORKINGTIME_n[3],
						POWERONCYCLES:=POWERONCYCLES_n[3],
						ENERGYCOUNTER:=ENERGYCOUNTER_n[3],
						ENERGYCOUNTER_t :=ENERGYCOUNTER_T_n[3],
						Lux_Enable => NODO03.w_DO_01,
						Lux_Auto:=NODO03.DI_01,
						Lux_Off:= NODO03.DI_02,
						Lux_Man:= NODO03.DI_03);

			(* CAMPATA 4 - CONTATORE N.5 *)

		IF   ZTHL04.ERR (*OR NODO04.Status_Log>0*) THEN
			BitStart04:=TRUE;
		ELSE
			IF ZTHL04.ValoreScalato <  SogliaLux04  THEN
				BitStart04:=TRUE;
			ELSIF   ZTHL04.ValoreScalato >   (LIMIT(0,SogliaLux04 + IsteresiLux04,ZTHL04.PuntoMaxX)) THEN
				BitStart04:=FALSE;
			END_IF;
		END_IF;
		ToffDelayLux4(IN:=BitStart04 AND CRON04.RunCrono, PT:= t#1s*delayOffLux, Q=> , ET=> );
		LuxElement04(DI_ONLux:=ToffDelayLux4.Q,
						Lux_State:=NODO04.DI_04,
						WORKINGTIME:=WORKINGTIME_n[4],
						POWERONCYCLES:=POWERONCYCLES_n[4],
						ENERGYCOUNTER:=ENERGYCOUNTER_n[4],
						ENERGYCOUNTER_t :=ENERGYCOUNTER_T_n[4],
						Lux_Enable => NODO04.w_DO_01,
						Lux_Auto:=NODO04.DI_01,
						Lux_Off:= NODO04.DI_02,
						Lux_Man:= NODO04.DI_03);

			(* CAMPATA 5 - CONTATORE N.6 *)

		IF   ZTHL05.ERR (*OR NODO05.Status_Log>0*) THEN
			BitStart05:=TRUE;
		ELSE
			IF ZTHL05.ValoreScalato <  SogliaLux05  THEN
				BitStart05:=TRUE;
			ELSIF   ZTHL05.ValoreScalato >   (LIMIT(0,SogliaLux05 + IsteresiLux05,ZTHL05.PuntoMaxX)) THEN
				BitStart05:=FALSE;
			END_IF;
		END_IF;
		ToffDelayLux5(IN:=BitStart05 AND CRON05.RunCrono, PT:= t#1s*delayOffLux, Q=> , ET=> );
		LuxElement05(DI_ONLux:=ToffDelayLux5.Q,
						Lux_State:=NODO05.DI_04,
						WORKINGTIME:=WORKINGTIME_n[5],
						POWERONCYCLES:=POWERONCYCLES_n[5],
						ENERGYCOUNTER:=ENERGYCOUNTER_n[5],
						ENERGYCOUNTER_t :=ENERGYCOUNTER_T_n[5],
						Lux_Enable => NODO05.w_DO_01,
						Lux_Auto:=NODO05.DI_01,
						Lux_Off:= NODO05.DI_02,
						Lux_Man:= NODO05.DI_03);

			(* CAMPATA 6 - CONTATORE N.7 *)

		IF   ZTHL06.ERR (*OR NODO06.Status_Log>0*) THEN
			BitStart06:=TRUE;
		ELSE
			IF ZTHL06.ValoreScalato <  SogliaLux06  THEN
				BitStart06:=TRUE;
			ELSIF   ZTHL06.ValoreScalato >  (LIMIT(0,SogliaLux06 + IsteresiLux06,ZTHL06.PuntoMaxX)) THEN
				BitStart06:=FALSE;

			END_IF;
		END_IF;
		ToffDelayLux6(IN:=BitStart06 AND CRON06.RunCrono, PT:= t#1s*delayOffLux, Q=> , ET=> );
		LuxElement06(DI_ONLux:=ToffDelayLux6.Q,
						Lux_State:=NODO06.DI_04,
						WORKINGTIME:=WORKINGTIME_n[6],
						POWERONCYCLES:=POWERONCYCLES_n[6],
						ENERGYCOUNTER:=ENERGYCOUNTER_n[6],
						ENERGYCOUNTER_t :=ENERGYCOUNTER_T_n[6],
						Lux_Enable => NODO06.w_DO_01,
						Lux_Auto:=NODO06.DI_01,
						Lux_Off:= NODO06.DI_02,
						Lux_Man:= NODO06.DI_03);

			(* CAMPATA 7 - CONTATORE N.8 *)

		IF   ZTHL07.ERR (*OR NODO07.Status_Log>0*) THEN
			BitStart07:=TRUE;
		ELSE
			IF ZTHL07.ValoreScalato <  SogliaLux07  THEN
				BitStart07:=TRUE;
			ELSIF   ZTHL07.ValoreScalato >  (LIMIT(0,SogliaLux07 + IsteresiLux07,ZTHL07.PuntoMaxX))  THEN
				BitStart07:=FALSE;
			END_IF;
		END_IF;

		ToffDelayLux7(IN:=BitStart07 AND CRON07.RunCrono, PT:= t#1s*delayOffLux, Q=> , ET=> );
		LuxElement07(DI_ONLux:=ToffDelayLux7.Q,
						Lux_State:=NODO07.DI_04,
						WORKINGTIME:=WORKINGTIME_n[7],
						POWERONCYCLES:=POWERONCYCLES_n[7],
						ENERGYCOUNTER:=ENERGYCOUNTER_n[7],
						ENERGYCOUNTER_t :=ENERGYCOUNTER_T_n[7],
						Lux_Enable => NODO07.w_DO_01,
						Lux_Auto:=NODO07.DI_01,
						Lux_Off:= NODO07.DI_02,
						Lux_Man:= NODO07.DI_03);


			(* CAMPATA 8 - CONTATORE N.9 *)

		IF   ZTHL08.ERR (*OR NODO08.Status_Log>0*) THEN
			BitStart08:=TRUE;
		ELSE
			IF ZTHL08.ValoreScalato <  SogliaLux08  THEN
				BitStart08:=TRUE;
			ELSIF   ZTHL08.ValoreScalato >   (LIMIT(0,SogliaLux08 + IsteresiLux08,ZTHL08.PuntoMaxX)) THEN
				BitStart08:=FALSE;
			END_IF;
		END_IF;
		ToffDelayLux8(IN:=BitStart08 AND CRON08.RunCrono, PT:= t#1s*delayOffLux, Q=> , ET=> );
		LuxElement08(DI_ONLux:=ToffDelayLux8.Q,
						Lux_State:=NODO08.DI_04,
						WORKINGTIME:=WORKINGTIME_n[8],
						POWERONCYCLES:=POWERONCYCLES_n[8],
						ENERGYCOUNTER:=ENERGYCOUNTER_n[8],
						ENERGYCOUNTER_t :=ENERGYCOUNTER_T_n[8],
						Lux_Enable => NODO08.w_DO_01,
						Lux_Auto:=NODO08.DI_01,
						Lux_Off:= NODO08.DI_02,
						Lux_Man:= NODO08.DI_03);

			(* CAMPATA 9 - CONTATORE N.10 *)

		IF   ZTHL09.ERR (*OR NODO09.Status_Log>0*) THEN
			BitStart09:=TRUE;
		ELSE
			IF ZTHL09.ValoreScalato <  SogliaLux09  THEN
				BitStart09:=TRUE;
			ELSIF   ZTHL09.ValoreScalato >  (LIMIT(0,SogliaLux09 + IsteresiLux09,ZTHL09.PuntoMaxX)) THEN
				BitStart09:=FALSE;
			END_IF;
		END_IF;
		ToffDelayLux9(IN:=BitStart09 AND CRON09.RunCrono, PT:= t#1s*delayOffLux, Q=> , ET=> );
		LuxElement09(DI_ONLux:=ToffDelayLux9.Q,
						Lux_State:=NODO09.DI_04,
						WORKINGTIME:=WORKINGTIME_n[9],
						POWERONCYCLES:=POWERONCYCLES_n[9],
						ENERGYCOUNTER:=ENERGYCOUNTER_n[9],
						ENERGYCOUNTER_t :=ENERGYCOUNTER_T_n[9],
						Lux_Enable => NODO09.w_DO_01,
						Lux_Auto:=NODO09.DI_01,
						Lux_Off:= NODO09.DI_02,
						Lux_Man:= NODO09.DI_03);

			(* MAGAZZINO - CONTATORE N.11 *)

		IF   ZTHL10.ERR (*OR NODO10.Status_Log>0*) THEN
			BitStart10:=TRUE;
		ELSE
			IF ZTHL10.ValoreScalato <  SogliaLux10  THEN
				BitStart10:=TRUE;
			ELSIF   ZTHL10.ValoreScalato >   (LIMIT(0,SogliaLux10 + IsteresiLux10,ZTHL10.PuntoMaxX)) THEN
				BitStart10:=FALSE;
			END_IF;
		END_IF;
		ToffDelayLux10(IN:=BitStart10 AND CRON10.RunCrono, PT:= t#1s*delayOffLux, Q=> , ET=> );
		LuxElement10(DI_ONLux:=ToffDelayLux10.Q,
						Lux_State:=NODO10.DI_04,
						WORKINGTIME:=WORKINGTIME_n[10],
						POWERONCYCLES:=POWERONCYCLES_n[10],
						ENERGYCOUNTER:=ENERGYCOUNTER_n[10],
						ENERGYCOUNTER_t :=ENERGYCOUNTER_T_n[10],
						Lux_Enable => NODO10.w_DO_01,
						Lux_Auto:=NODO10.DI_01,
						Lux_Off:= NODO10.DI_02,
						Lux_Man:= NODO10.DI_03);

			(* CAMPATA 1-2 - EMERGENZA  *)

		IF   ZTHL02.ERR (*OR NODO02.Status_Log>0*) THEN
			BitStart11:=TRUE;
		ELSE
			IF ZTHL02.ValoreScalato <  SogliaLux11  THEN
				BitStart11:=TRUE;
			ELSIF   ZTHL02.ValoreScalato >   (LIMIT(0,SogliaLux11 + IsteresiLux11,ZTHL02.PuntoMaxX)) THEN
				BitStart11:=FALSE;
			END_IF;
		END_IF;
		ToffDelayLux11(IN:=BitStart11 , PT:= t#1s*delayOffLux, Q=> , ET=> );
		LuxElement11(DI_ONLux:=ToffDelayLux11.Q,
						Lux_State:=ToffDelayLux11.Q,   (* Non ha Feedback *)
						WORKINGTIME:=WORKINGTIME_n[11],
						POWERONCYCLES:=POWERONCYCLES_n[11],
						ENERGYCOUNTER:=ENERGYCOUNTER_n[11],
						ENERGYCOUNTER_t :=ENERGYCOUNTER_T_n[11],
						Lux_Enable => NODO02.w_DO_02,
						Lux_Auto:=NODO02.DI_01,
						Lux_Off:= NODO02.DI_02,
						Lux_Man:= NODO02.DI_03);

			(* CAMPATA 3 - EMERGENZA  *)

		IF   ZTHL03.ERR (*OR NODO03.Status_Log>0*) THEN
			BitStart12:=TRUE;
		ELSE
			IF ZTHL03.ValoreScalato <  SogliaLux12  THEN
				BitStart12:=TRUE;
			ELSIF   ZTHL03.ValoreScalato >   (LIMIT(0,SogliaLux12 + IsteresiLux12,ZTHL03.PuntoMaxX)) THEN
				BitStart12:=FALSE;

			END_IF;
		END_IF;
		ToffDelayLux12(IN:=BitStart12 , PT:= t#1s*delayOffLux, Q=> , ET=> );
		LuxElement12(DI_ONLux:=ToffDelayLux12.Q,
						Lux_State:=ToffDelayLux12.Q,   (* Non ha Feedback *)
						WORKINGTIME:=WORKINGTIME_n[12],
						POWERONCYCLES:=POWERONCYCLES_n[12],
						ENERGYCOUNTER:=ENERGYCOUNTER_n[12],
						ENERGYCOUNTER_t :=ENERGYCOUNTER_T_n[12],
						Lux_Enable => NODO03.w_DO_02,
						Lux_Auto:=NODO03.DI_01,
						Lux_Off:= NODO03.DI_02,
						Lux_Man:= NODO03.DI_03);







			CASE IndiceAnz OF

					1:typeVisuANZ:=ANZ01.measures;
					2:typeVisuANZ:=ANZ02.measures;
					3:typeVisuANZ:=ANZ03.measures;
					4:typeVisuANZ:=ANZ04.measures;
					5:typeVisuANZ:=ANZ05.measures;
					6:typeVisuANZ:=ANZ06.measures;
					7:typeVisuANZ:=ANZ07.measures;
					8:typeVisuANZ:=ANZ08.measures;
					9:typeVisuANZ:=ANZ09.measures;
					10:typeVisuANZ:=ANZ10.measures;
					11:typeVisuANZ:=ANZ11.measures;
			ELSE
					IndiceAnz:=1;
			END_CASE;



						VisuTestoANZ[1,1]:='COSPHI_L1';
						VisuTestoANZ[1,2]:='COSPHI_L2';
						VisuTestoANZ[1,3]:='COSPHI_L3';
						VisuTestoANZ[1,4]:='FREQ';
						VisuTestoANZ[1,5]:='I_L1';
						VisuTestoANZ[1,6]:='I_L1_Max';
						VisuTestoANZ[1,7]:='I_L2';
						VisuTestoANZ[1,8]:='I_L2_Max';
						VisuTestoANZ[1,9]:='I_L3';
						VisuTestoANZ[1,10]:='I_L3_Max';
						VisuTestoANZ[1,11]:='P_3P';
						VisuTestoANZ[1,12]:='P_3P_Avg';
						VisuTestoANZ[1,13]:='P_3P_max';
						VisuTestoANZ[1,14]:='PF_L1';
						VisuTestoANZ[1,15]:='PF_L2';
						VisuTestoANZ[1,16]:='PF_L3';
						VisuTestoANZ[1,17]:='Q_3P';
						VisuTestoANZ[1,18]:='Q_3P_Max';
						VisuTestoANZ[1,19]:='V_L1L2';
						VisuTestoANZ[1,20]:='V_L1N';
						VisuTestoANZ[1,21]:='V_L2L3';
						VisuTestoANZ[1,22]:='V_L3N';
						VisuTestoANZ[1,23]:='V_L3L1';
						VisuTestoANZ[1,24]:='V_L3N';
						VisuTestoANZ[1,25]:='WH_3P';
						VisuTestoANZ[1,26]:='VARH_3P';





						VisuTestoANZ[2,1]:=REAL_TO_STRING(typeVisuANZ.COSPHI_L1);
						VisuTestoANZ[2,2]:=REAL_TO_STRING(typeVisuANZ.COSPHI_L2);
						VisuTestoANZ[2,3]:=REAL_TO_STRING(typeVisuANZ.COSPHI_L3);
						VisuTestoANZ[2,4]:=REAL_TO_STRING(typeVisuANZ.FREQ);
						VisuTestoANZ[2,5]:=REAL_TO_STRING(typeVisuANZ.I_L1);
						VisuTestoANZ[2,6]:=REAL_TO_STRING(typeVisuANZ.I_L1_Max);
						VisuTestoANZ[2,7]:=REAL_TO_STRING(typeVisuANZ.I_L2);
						VisuTestoANZ[2,8]:=REAL_TO_STRING(typeVisuANZ.I_L2_Max);
						VisuTestoANZ[2,9]:=REAL_TO_STRING(typeVisuANZ.I_L3);
						VisuTestoANZ[2,10]:=REAL_TO_STRING(typeVisuANZ.I_L3_Max);
						VisuTestoANZ[2,11]:=REAL_TO_STRING(typeVisuANZ.P_3P);
						VisuTestoANZ[2,12]:=REAL_TO_STRING(typeVisuANZ.P_3P_Avg);
						VisuTestoANZ[2,13]:=REAL_TO_STRING(typeVisuANZ.P_3P_max);;
						VisuTestoANZ[2,14]:=REAL_TO_STRING(typeVisuANZ.PF_L1);
						VisuTestoANZ[2,15]:=REAL_TO_STRING(typeVisuANZ.PF_L2);
						VisuTestoANZ[2,16]:=REAL_TO_STRING(typeVisuANZ.PF_L3);
						VisuTestoANZ[2,17]:=REAL_TO_STRING(typeVisuANZ.Q_3P);
						VisuTestoANZ[2,18]:=REAL_TO_STRING(typeVisuANZ.Q_3P_Max);
						VisuTestoANZ[2,19]:=REAL_TO_STRING(typeVisuANZ.V_L1L2);
						VisuTestoANZ[2,20]:=REAL_TO_STRING(typeVisuANZ.V_L1N);
						VisuTestoANZ[2,21]:=REAL_TO_STRING(typeVisuANZ.V_L2L3);
						VisuTestoANZ[2,22]:=REAL_TO_STRING(typeVisuANZ.V_L3N);
						VisuTestoANZ[2,23]:=REAL_TO_STRING(typeVisuANZ.V_L3L1);
						VisuTestoANZ[2,24]:=REAL_TO_STRING(typeVisuANZ.V_L3N);
						VisuTestoANZ[2,25]:=REAL_TO_STRING(typeVisuANZ.WH_3P);
						VisuTestoANZ[2,26]:=REAL_TO_STRING(typeVisuANZ.VARH_3P);





			Lamp( Allarme:=ZTHL01.Status_Log=2 OR
  						  	ZTHL02.Status_Log=2 OR
  						  	ZTHL03.Status_Log=2 OR
  						  	ZTHL04.Status_Log=2 OR
 						  	ZTHL05.Status_Log=2 OR
						  	ZTHL06.Status_Log=2 OR
						  	ZTHL07.Status_Log=2 OR
						  	ZTHL08.Status_Log=2 OR
						  	ZTHL09.Status_Log=2 OR
						  	ZTHL10.Status_Log=2 OR
							ANZ01.Status_Log=2 OR
							ANZ02.Status_Log=2 OR
							ANZ03.Status_Log=2 OR
							ANZ04.Status_Log=2 OR
							ANZ05.Status_Log=2 OR
							ANZ06.Status_Log=2 OR
							ANZ07.Status_Log=2 OR
							ANZ08.Status_Log=2 OR
							ANZ09.Status_Log=2 OR
							ANZ10.Status_Log=2 OR
							ANZ11.Status_Log=2 OR
							NODO01.Status_Log=2 OR
							NODO02.Status_Log=2 OR
							NODO03.Status_Log=2 OR
							NODO04.Status_Log=2 OR
							NODO05.Status_Log=2 OR
							NODO06.Status_Log=2 OR
							NODO07.Status_Log=2 OR
							NODO08.Status_Log=2 OR
							NODO09.Status_Log=2 OR
							NODO10.Status_Log=2
							,
							Warning:=	ZTHL01.Status_Log=1 OR
  						  	ZTHL02.Status_Log=1 OR
  						  	ZTHL03.Status_Log=1 OR
  						  	ZTHL04.Status_Log=1 OR
 						  	ZTHL05.Status_Log=1 OR
						  	ZTHL06.Status_Log=1 OR
						  	ZTHL07.Status_Log=1 OR
						  	ZTHL08.Status_Log=1 OR
						  	ZTHL09.Status_Log=1 OR
						  	ZTHL10.Status_Log=1 OR
							ANZ01.Status_Log=1 OR
							ANZ02.Status_Log=1 OR
							ANZ03.Status_Log=1 OR
							ANZ04.Status_Log=1 OR
							ANZ05.Status_Log=1 OR
							ANZ06.Status_Log=1 OR
							ANZ07.Status_Log=1 OR
							ANZ08.Status_Log=1 OR
							ANZ09.Status_Log=1 OR
							ANZ10.Status_Log=1 OR
							ANZ11.Status_Log=1 OR
							NODO01.Status_Log=1 OR
							NODO02.Status_Log=1 OR
							NODO03.Status_Log=1 OR
							NODO04.Status_Log=1 OR
							NODO05.Status_Log=1 OR
							NODO06.Status_Log=1 OR
							NODO07.Status_Log=1 OR
							NODO08.Status_Log=1 OR
							NODO09.Status_Log=1 OR
							NODO10.Status_Log=1
							,
							AllarmeLampada=>LAMP_AL
							);

			(* Test toggle *)
		(*	IF TEST1 THEN TEST1:=FALSE; ELSE TEST1:=TRUE; END_IF*)
		END_IF





		Timer3(IN:=NOT Timer3.Q,PT:=T#5m);

		R_TrigAggiornaLog(clk:=(Timer3.Q OR RichiestaDaRemoto OR HMI_AggiornaLog) );

		IF R_TrigAggiornaLog.Q AND loggando=FALSE  THEN
			(* Trig logger *)
		(*	LogTrig(); *)
			EseguiLog:=10;
			loggando:=TRUE;
	     END_IF

	CASE Eseguilog  OF

			10 : 	Ton_pausaTrig(IN:=FALSE , PT:=TempoLog , Q=> , ET=> );
					Logger_Head();

						ANZ01.AddLogData();
						ANZ02.AddLogData();
						ANZ03.AddLogData();
						ANZ04.AddLogData();
						ANZ05.AddLogData();
					Logger_Send();
					EseguiLog:=15;

			15: Ton_pausaTrig(IN:=TRUE , PT:=TempoLog , Q=> , ET=> );
					IF Ton_pausaTrig.Q THEN
						EseguiLog:=20;
					END_IF

			20 : 	Ton_pausaTrig(IN:=FALSE , PT:=TempoLog , Q=> , ET=> );
					Logger_Head();
					ANZ06.AddLogData();
					ANZ07.AddLogData();
					ANZ08.AddLogData();
					ANZ09.AddLogData();
					ANZ10.AddLogData();
					ANZ11.AddLogData();


					Logger_Send();
					EseguiLog:=25;

			25: Ton_pausaTrig(IN:=TRUE , PT:=TempoLog , Q=> , ET=> );
					IF Ton_pausaTrig.Q THEN
						EseguiLog:=30;
					END_IF

			30 : 	Ton_pausaTrig(IN:=FALSE , PT:=TempoLog , Q=> , ET=> );
					Logger_Head();
					ZTHL01.AddLogData();
					ZTHL02.AddLogData();
					ZTHL03.AddLogData();
					ZTHL04.AddLogData();
					ZTHL05.AddLogData();
					Logger_Send();
					EseguiLog:=35;
			35: Ton_pausaTrig(IN:=TRUE , PT:=TempoLog , Q=> , ET=> );
					IF Ton_pausaTrig.Q THEN
						EseguiLog:=36;
					END_IF
			36 : 	Ton_pausaTrig(IN:=FALSE , PT:=TempoLog , Q=> , ET=> );
					Logger_Head();
					ZTHL06.AddLogData();
					ZTHL07.AddLogData();
					ZTHL08.AddLogData();
					ZTHL09.AddLogData();
					ZTHL10.AddLogData();
					Logger_Send();
					EseguiLog:=40;

			40: Ton_pausaTrig(IN:=TRUE , PT:=TempoLog, Q=> , ET=> );
					IF Ton_pausaTrig.Q THEN
						EseguiLog:=50;
					END_IF

			50 : 	Ton_pausaTrig(IN:=FALSE , PT:=TempoLog , Q=> , ET=> );
					Logger_Head();
					CRON01.AddLogData();
					CRON02.AddLogData();
					CRON03.AddLogData();
					CRON04.AddLogData();
					CRON05.AddLogData();
					CRON06.AddLogData();
					CRON07.AddLogData();
					CRON08.AddLogData();
					CRON09.AddLogData();
					CRON10.AddLogData();

					Logger_Send();
					EseguiLog:=60;

			60: Ton_pausaTrig(IN:=TRUE , PT:=TempoLog, Q=> , ET=> );
					IF Ton_pausaTrig.Q THEN
						EseguiLog:=70;
					END_IF

			70 : 	Ton_pausaTrig(IN:=FALSE , PT:=TempoLog , Q=> , ET=> );
					Logger_Head();
					LuxElement01.AddLogData(WORKINGTIME:=WORKINGTIME_n[1],POWERONCYCLES:=POWERONCYCLES_n[1],ENERGYCOUNTER:=ENERGYCOUNTER_n[1],
												ENERGYCOUNTER_t :=ENERGYCOUNTER_T_n[1]);
					LuxElement02.AddLogData(WORKINGTIME:=WORKINGTIME_n[1],POWERONCYCLES:=POWERONCYCLES_n[1],ENERGYCOUNTER:=ENERGYCOUNTER_n[1],
												ENERGYCOUNTER_t :=ENERGYCOUNTER_T_n[1]);
					LuxElement03.AddLogData(WORKINGTIME:=WORKINGTIME_n[1],POWERONCYCLES:=POWERONCYCLES_n[1],ENERGYCOUNTER:=ENERGYCOUNTER_n[1],
												ENERGYCOUNTER_t :=ENERGYCOUNTER_T_n[1]);
					LuxElement04.AddLogData(WORKINGTIME:=WORKINGTIME_n[1],POWERONCYCLES:=POWERONCYCLES_n[1],ENERGYCOUNTER:=ENERGYCOUNTER_n[1],
												ENERGYCOUNTER_t :=ENERGYCOUNTER_T_n[1]);
					LuxElement05.AddLogData(WORKINGTIME:=WORKINGTIME_n[1],POWERONCYCLES:=POWERONCYCLES_n[1],ENERGYCOUNTER:=ENERGYCOUNTER_n[1],
												ENERGYCOUNTER_t :=ENERGYCOUNTER_T_n[1]);
					LuxElement06.AddLogData(WORKINGTIME:=WORKINGTIME_n[1],POWERONCYCLES:=POWERONCYCLES_n[1],ENERGYCOUNTER:=ENERGYCOUNTER_n[1],
												ENERGYCOUNTER_t :=ENERGYCOUNTER_T_n[1]);
					LuxElement07.AddLogData(WORKINGTIME:=WORKINGTIME_n[1],POWERONCYCLES:=POWERONCYCLES_n[1],ENERGYCOUNTER:=ENERGYCOUNTER_n[1],
												ENERGYCOUNTER_t :=ENERGYCOUNTER_T_n[1]);
					LuxElement08.AddLogData(WORKINGTIME:=WORKINGTIME_n[1],POWERONCYCLES:=POWERONCYCLES_n[1],ENERGYCOUNTER:=ENERGYCOUNTER_n[1],
												ENERGYCOUNTER_t :=ENERGYCOUNTER_T_n[1]);
					LuxElement09.AddLogData(WORKINGTIME:=WORKINGTIME_n[1],POWERONCYCLES:=POWERONCYCLES_n[1],ENERGYCOUNTER:=ENERGYCOUNTER_n[1],
												ENERGYCOUNTER_t :=ENERGYCOUNTER_T_n[1]);
					LuxElement10.AddLogData(WORKINGTIME:=WORKINGTIME_n[1],POWERONCYCLES:=POWERONCYCLES_n[1],ENERGYCOUNTER:=ENERGYCOUNTER_n[1],
												ENERGYCOUNTER_t :=ENERGYCOUNTER_T_n[1]);
					LuxElement11.AddLogData(WORKINGTIME:=WORKINGTIME_n[1],POWERONCYCLES:=POWERONCYCLES_n[1],ENERGYCOUNTER:=ENERGYCOUNTER_n[1],
												ENERGYCOUNTER_t :=ENERGYCOUNTER_T_n[1]);
					LuxElement12.AddLogData(WORKINGTIME:=WORKINGTIME_n[1],POWERONCYCLES:=POWERONCYCLES_n[1],ENERGYCOUNTER:=ENERGYCOUNTER_n[1],
												ENERGYCOUNTER_t :=ENERGYCOUNTER_T_n[1]);


					Logger_Send();
					EseguiLog:=200;




			200:
				RichiestaDaRemoto:=FALSE;
				loggando:=FALSE;
				RichiestaDaRemoto:=FALSE;

		END_CASE







	S_SHUTDOWN:
		(* Stop caldaia *)
		(* Stop deviatori *)
		(* Aspetta 5 min prima di spegnere eventuali circolatori *)
		Sys.Status:=S_STARTUP;

	S_HALT:
		(* Aspetta uscita manuale *)
		Sys.Status:=S_STARTUP;


ELSE
	Sys.Status:=S_STARTUP;
END_CASE;
END_ACTION

(* POU TCP_Logger/Logger_Proc, ST *)
PROGRAM Logger_Proc
VAR
	c1:         	TCPCLIENT;

	Open:	    	BOOL;
	IpAddr:			DWORD;
	InetAddr:		DWORD;
	Connected:  	BOOL;
	Error:      	DINT;
	TxTrig:     	BOOL;
	RxData:			ARRAY [0..MAX_RECEIVE_TCP_CLIENT] OF BYTE;
	RxLen:			DINT;

	Retry:			BYTE;	(* Counter for connection retries *)
	Recovered:		BYTE;	(* Counter for recovered unsent messages *)

	i:				DINT;
	pos:			DWORD;
	hFile:			DWORD;

END_VAR
(*=== State machine ===*)
CASE Logger.Status OF

	S_Logger_UNKNOWN:
		(* Startup *)
		Logger.SendReq:=FALSE;
		Open:=FALSE;
		Logger.Status:=S_Logger_IDLE;

	S_Logger_IDLE:
		(* Wait request *)
		IF Logger.SendReq THEN
			(* Resolve server name or use static IP *)
			IF LEN(Logger_SERVER)=0 THEN
				InetAddr:=SysSockInetAddr(Logger_IP);
			ELSE
				IpAddr:=SysSockGetHostByName(ADR(Logger_SERVER));
				DWORDSWAP(pIn:=ADR(IpAddr), pOut:=ADR(InetAddr));
			END_IF
			TxTrig:=FALSE;
			RxLen:=0;
			(* Open connection *)
			Open:=TRUE;
			Logger.Status:=S_Logger_WAITCONN;
		END_IF

	S_Logger_WAITCONN:
		(* Wait connection *)
		IF Connected THEN
			(* Send data *)
			TxTrig:=TRUE;
			Logger.Status:=S_Logger_WAITTX;
		END_IF
		IF Error>0 THEN
			Open:=FALSE;
			Logger.Status:=S_Logger_ERROR;
		END_IF

	S_Logger_WAITTX:
		(* Wait transmission *)
		IF NOT TxTrig THEN
			Logger.Status:=S_Logger_WAITRESP;
		END_IF
		IF Error>0 THEN
			Open:=FALSE;
			Logger.Status:=S_Logger_ERROR;
		END_IF

	S_Logger_WAITRESP:
		(* Wait response *)
		IF Connected=FALSE (* OR TIMEOUT!! *) THEN
			Open:=FALSE;
			(* Check response *)
			(*--diego*)
			(* Check unsent messages to flush *)
				IF Recovered<Logger_RecoverMsgs THEN
					MsgChk();
					IF Logger.SendReq=TRUE THEN
						Recovered:=Recovered+1;
					ELSE
						Recovered:=0;
					END_IF
				ELSE
					Recovered:=0;
				END_IF
				Logger.Status:=S_Logger_IDLE;
			(*--diego--*)
			IF RxLen>=4 AND CHKSTRING(pString:=ADR(RxData), pPattern:=ADR(Logger_CHECK)) THEN
				Logger.SendReq:=FALSE;
				Retry:=0;
				(* Check unsent messages to flush *)
				IF Recovered<Logger_RecoverMsgs THEN
					MsgChk();
					IF Logger.SendReq=TRUE THEN
						Recovered:=Recovered+1;
					ELSE
						Recovered:=0;
					END_IF
				ELSE
					Recovered:=0;
				END_IF
				Logger.Status:=S_Logger_IDLE;
			ELSE
				Logger.Status:=S_Logger_ERROR;
			END_IF
		END_IF

	S_Logger_ERROR:
		(* Connection error or send failure *)
		Retry:=Retry+1;
		IF Retry>Logger_ConnRetries THEN
			(* Save message as unsent *)
			MsgSave();
			Logger.SendReq:=FALSE;
			Retry:=0;
		END_IF
		Logger.Status:=S_Logger_IDLE;

ELSE
	Logger.Status:=S_Logger_UNKNOWN;
END_CASE


(*=== Execute client lib ===*)
c1(
	xOpenConnection			:= Open,
	dwInetAddr 				:= InetAddr,
	wPortNumber				:= Logger_PORT,
	ptSendData				:= ADR(Logger.SendData),
	diSendCount				:= Logger.SendLen,
	tConnectWatchdogTime	:= t#10s,
	xStartSend				:= TxTrig,
	aReceiveBuffer			:= RxData,
	diReceiveCount			:= RxLen,
	xConnected				=> Connected,
	diError					=> Error
);

(*=== Process Rx data ===*)
(*IF RxLen>0 THEN
	RxLen:=0;
END_IF*)
END_PROGRAM
ACTION MsgChk:
(* Open index file *)
hFile:=SysFileOpen(Logger_IndexFile,'r');
IF hFile=0 THEN
	RETURN;
END_IF
(* Search oldest message to recover *)
SysFileSetPos(hFile,Logger.LastIdxPos);
Logger.SendLen:=0;
REPEAT
	SysFileRead(hFile, ADR(Logger.SendIdx), SIZEOF(Logger.SendIdx));
	pos:=SysFileGetPos(hFile);
	SysFileRead(hFile, ADR(Logger.SendLen), SIZEOF(Logger.SendLen));
UNTIL
	SysFileEOF(hFile) OR Logger.SendLen<>0
END_REPEAT
SysFileClose(hFile);
(* Delete index file when all messages are recovered *)
IF Logger.SendLen=0 THEN
	Logger.LastIdxPos:=0;
	SysFileDelete(Logger_IndexFile);
	RETURN;
END_IF
(* Recover message data *)
hFile:=SysFileOpen(Logger_DataFile,'r');
IF hFile<>0 THEN
	SysFileSetPos(hFile,Logger.SendIdx);
	SysFileRead(hFile,ADR(Logger.SendData),Logger.SendLen);
	Logger.SendReq:=TRUE;
	SysFileClose(hFile);
END_IF
(* Clear index entry *)
hFile:=SysFileOpen(Logger_IndexFile,'a');
IF hFile<>0 THEN
	SysFileSetPos(hFile,pos);
	i:=0;
	SysFileWrite(hFile, ADR(i), 4);
	Logger.LastIdxPos:=SysFileGetPos(hFile);
	SysFileClose(hFile);
END_IF
END_ACTION
ACTION MsgSave:
(* Add log position in recovery indexes *)
hFile:=SysFileOpen(Logger_IndexFile,'a');
SysFileWrite(hFile, ADR(Logger.SendIdx), SIZEOF(Logger.SendIdx));
SysFileWrite(hFile, ADR(Logger.SendLen), SIZEOF(Logger.SendLen));
SysFileClose(hFile);
END_ACTION

(* POU Utils Functions/TCPCLIENT, ST *)
FUNCTION_BLOCK TCPCLIENT
(***********************************************************************************************************	*)
(* Version: 1.3b                        			          													*)
(* Date: 28.10.2014                   				          							            			*)
(***********************************************************************************************************	*)
(* WAGO Kontakttechnik GmbH Hansastr. 27 32423 Minden(Westf.)													*)
(* Tel. +0049 571/887-0 Fax. +0049 571/887-0																	*)
(* Author: VB																									*)
(***********************************************************************************************************	*)
(*Description:	A TCP client to read and write data with additional connection watchdog							*)
(*History:																										*)
(*Version 1.3b: 28.10.2014: Use DWORD address for IP (Andrea Ravasio)											*)
(*Version 1.3: 11.02.2011: Changes according to 750-880/881											 			*)
(*Version 1.2: 29.08.2007 Bugfix TCP Client																		*)
(*Version 1.1: 15.01.2007 Changes according to FW11																*)
(*Version 1.0: 09.03.2006 Release																				*)
(***********************************************************************************************************	*)
VAR CONSTANT
	STATE_CREATE     				 : BYTE:= 0;
	STATE_OPEN     					 : BYTE:= 1;
	STATE_IOCTL    					 : BYTE:= 2;
	STATE_CONNECT     				 : BYTE:= 10;
	STATE_TX       					 : BYTE:= 20;
	STATE_RX       					 : BYTE:= 30;
	STATE_CLOSE    					 : BYTE:= 40;
	STATE_ERROR_TRAP			     : BYTE:= 200;
END_VAR

VAR_INPUT
	xOpenConnection					: BOOL;
	dwInetAddr						: DWORD; (* <== Use SysSockInetAddr() value or
													swapped bytes order of SysSockGetHostByName() value *)
	wPortNumber						: WORD;
	ptSendData						: POINTER TO ARRAY[0..MAX_SEND_TCP_CLIENT] OF BYTE;
	diSendCount						: DINT;
	tConnectWatchdogTime		    : TIME := t#10s;
END_VAR
VAR_OUTPUT
	xConnected						: BOOL;
	diError 						: DINT := 0;
END_VAR
(* ErrorCodes -----------------------------------------
	16#8001 => No socket descriptor available 
	16#8002 => SysSockSend returns -1 
	16#8003 => Socket was "gracefully closed" 
	16#8004 => switching to none blocking mode fails
	16#8005 => SysSockClose() returns FALSE 
    16#8006 => SysSockConnect() fails
    16#8007 => SysSockSend() fails
	16#8008 => error state machine 
	16#8009 => timeout while waiting for data from server 
------------------------------------------------------------*)
VAR_IN_OUT
	xStartSend							: BOOL;
	aReceiveBuffer						: ARRAY [0..MAX_RECEIVE_TCP_CLIENT] OF BYTE;
	diReceiveCount						: DINT;
END_VAR
VAR
	m_State								: BYTE := 0;
	m_ReceiveBuffer						: ARRAY [0..MAX_RECEIVE_TCP_CLIENT_SOCKET] OF BYTE;
	m_Socket							: DINT;
	m_AddressInfo						: SOCKADDRESS;
	m_BytesReceived						: DINT;
	m_diReturn							: DINT;
	m_xReturn							: BOOL;
	m_IoCtlParameter  					: DINT := 1; (* IOCTL-Parameter for non-blocking mode of sockets *)
	i									: INT;
	T_Connect							: TON;
	m_count								: DINT;
	diOption							: DINT := 1;
	m_Blocking   						: DINT := 0;
END_VAR
IF xOpenConnection THEN
	(* State maschine *)
	CASE  m_State OF

	(* -------------------------------------------------------------------------*)
	STATE_CREATE:
			(* create socket descriptor*)
			m_Socket := SysSockCreate(diAddressFamily	:= SOCKET_AF_INET,
													 diType		:= SOCKET_STREAM,
													 diProtocol := SOCKET_IPPROTO_TCP);
			IF m_Socket >= 0 THEN
			(*Set Push-Bit*)
				IF ADR(%MW0)=16#30000000  OR ADR(%MW0)=16#20000000 THEN (*841 or 881*)
					SysSockSetOption(
						diSocket:=m_Socket,
						diLevel:=6,
						diOption:=SOCKET_TCP_NODELAY,
						pOptionValue:=ADR(diOption),
						diOptionLength:=SIZEOF(diOption));
				ELSE
						;
				END_IF
				m_State := STATE_IOCTL; (* succesful *)
			ELSE
				diError := 16#8001;  (* no socket descriptor available *)
				m_State := STATE_ERROR_TRAP;
			END_IF

	(* -------------------------------------------------------------------------*)
	STATE_IOCTL: (* change  socket mode  to none blocking *)
		m_diReturn := SysSockIoctl( m_Socket, SOCKET_FIONBIO, ADR(m_IoCtlParameter));
		IF m_diReturn <> 0 THEN
			m_AddressInfo.sin_family := SOCKET_AF_INET;
			m_AddressInfo.sin_port := SysSockNtohs(wPortNumber);
			m_AddressInfo.sin_addr := dwInetAddr;
			m_State := STATE_CONNECT;
		ELSE
			diError := 16#8004;  (* switching to none blocking mode fails *)
			m_State := STATE_ERROR_TRAP;
		END_IF


	(* -------------------------------------------------------------------------*)
	STATE_CONNECT: (* connect with server *)
		T_Connect(IN:=TRUE , PT:=tConnectWatchdogTime);(*activate watchdog for establishing connection to a server*)
		m_xReturn := SysSockConnect ( m_Socket, ADR(m_AddressInfo),  SIZEOF(m_AddressInfo));
		IF m_xReturn THEN (* succesful *)
			IF xStartSend THEN
				m_State := STATE_TX;(*transmit data*)
			ELSE
				m_State := STATE_RX;(*wait for data from server*)
			END_IF
			xConnected:=TRUE;
			T_Connect(IN:=FALSE);
		ELSE
			IF T_Connect.Q THEN
				diError := 16#8006;  (* connect fails *)
				xConnected:=FALSE;
				T_Connect(IN:=FALSE);
				m_State := STATE_ERROR_TRAP;
				SysSockClose( m_Socket);
			ELSE
				m_State := STATE_CONNECT;(*client still  tries to set up connection*)
			END_IF
		END_IF


	STATE_TX:	 (* send TCP-message *)
		m_diReturn := SysSockSend(diSocket := m_Socket,
								  pbyBuffer := ADR(ptSendData^[0]),
								  diBufferSize := diSendCount-m_count,
								  diFlags := 0);

		CASE m_diReturn OF
		-1:	(* ERROR *)
			T_Connect(IN:=TRUE , PT:=CONNECT_WATCHDOG_TIME);(*activate watchdog to check communication*)
			IF t_Connect.Q THEN
				diError := 16#8007;
				T_Connect(IN:=FALSE);
				m_State:=STATE_CLOSE;
			END_IF
		0: (* socket was "gracefully closed" *)
			m_State := STATE_CLOSE;
			diError := 16#8003;
		ELSE (* succesful *)
			m_count:=m_count+m_diReturn;
			IF m_count>=diSendCount THEN
				diError := 16#0000;
				m_State := STATE_RX;
				m_count:=0;
				xStartSend:=FALSE;
			END_IF
			T_Connect(IN:=FALSE);
		END_CASE

	(* -------------------------------------------------------------------------*)
	STATE_RX: (* process receive data *)
			m_BytesReceived := SysSockRecv(	diSocket 	:= m_Socket,
										pbyBuffer 	:= ADR(m_ReceiveBuffer),		(* Address of receive buffer *)
										diBufferSize:= SIZEOF(m_ReceiveBuffer),
										diFlags		:= 0);

			CASE m_BytesReceived OF
			-1:	(* No data available or error occured *)
				T_Connect(IN:=TRUE , PT:=tConnectWatchdogTime);(*activate watchdog to check communication*)
				IF t_Connect.Q THEN
					diError:=16#8009;
					T_Connect(IN:=FALSE);
					m_State:=STATE_CLOSE;
				END_IF
				IF xStartSend THEN
					m_State:=STATE_TX	;(* WAIT IN THIS STATE  and check for arriving data or new send command*)
				END_IF;
			0: (* socket was "gracefully closed"  *)
				m_State:=STATE_CLOSE;
				diError := 16#8003;
			ELSE (* succesful *)
				diError := 16#0000;
				T_Connect(IN:=FALSE);
				(* Copy received data into receive buffer *)
				FOR i:= 0 TO DINT_TO_INT(m_BytesReceived	)-1 DO
					aReceiveBuffer[diReceiveCount]:= m_ReceiveBuffer[i];
					diReceiveCount:=(diReceiveCount+1) MOD SIZEOF(aReceiveBuffer);
				END_FOR

			END_CASE

	(* -------------------------------------------------------------------------*)
	STATE_CLOSE : (* close socket *)
		IF ADR(%MW0)=16#30000000  OR ADR(%MW0)=16#20000000 THEN (*841 or 881*)
			;
		ELSE
			SysSockShutdown(m_Socket, 0);;(*870*)
		END_IF
		m_xReturn := SysSockClose( m_Socket);
		m_Socket := -1;
		m_State := 0; (* succesful *)
		xConnected:=FALSE;
		T_Connect(IN:=FALSE);
	(* -------------------------------------------------------------------------*)
	STATE_ERROR_TRAP: (* error handling *)
		xConnected:=FALSE;

	ELSE  (* Bad FSM code trap  *)
			m_State:= STATE_ERROR_TRAP;
			diError:= 16#8008;
	END_CASE

ELSE(*close connection*)
	IF m_Socket >= 0 THEN
		IF ADR(%MW0)=16#30000000  OR ADR(%MW0)=16#20000000 THEN (*841 or 881*)
			;
		ELSE
			SysSockShutdown(m_Socket, 0);;(*870*)
		END_IF
		SysSockClose( m_Socket);
	END_IF
	m_Socket := -1;
	diError := 16#0000;
	m_State := STATE_CREATE;
	xConnected:=FALSE;
	T_Connect(IN:=FALSE);
END_IF
END_FUNCTION_BLOCK

(* POU Utils Functions/DWORDSWAP, ST *)
FUNCTION DWORDSWAP:BOOL
VAR_INPUT
	pIn:POINTER TO ARRAY[1..4] OF BYTE;
	pOut:POINTER TO ARRAY[1..4] OF BYTE;
END_VAR
VAR
END_VAR
pOut^[1]:=pIn^[4];
pOut^[2]:=pIn^[3];
pOut^[3]:=pIn^[2];
pOut^[4]:=pIn^[1];
END_FUNCTION

(* POU Utils Functions/CHKSTRING, ST *)
FUNCTION CHKSTRING : BOOL
VAR_INPUT
	pString: POINTER TO BYTE;
	pPattern: POINTER TO BYTE;
END_VAR
VAR
END_VAR
CHKSTRING:=TRUE;
WHILE pPattern^<>0 AND CHKSTRING DO
	IF pPattern^<>pString^ THEN CHKSTRING:=FALSE; END_IF
	pString:=pString+1;
	pPattern:=pPattern+1;
END_WHILE
END_FUNCTION

(* POU TCP_Remote/Remote_Proc, ST *)
PROGRAM Remote_Proc
VAR
	s1:         	TCPSERVER;
	Enable: 		BOOL;
	Connected: 		BOOL;
	Error: 			DINT;

	TxData:			ARRAY[0..MAX_SEND_TCP_SERVER] OF BYTE;
	TxLen:			DINT;
	TxTrig:			BOOL;

	RxData:			ARRAY [0..MAX_RECEIVE_TCP_SERVER] OF BYTE;
	RxLen:			DINT;

	Status:			DINT;

	(* Command interpreter *)

	Cmd_Buf:		ARRAY [0..MAX_RECEIVE_TCP_SERVER] OF BYTE;
	Cmd_Buf_U16:	POINTER TO WORD;
	Cmd_Buf_INT:	POINTER TO INT;
	Cmd_BufLen:		WORD;
	Cmd_St:			WORD;

	Cmd_Obj:		WORD;
	Cmd_ObjIdx:		WORD;
	Cmd_C:			WORD;
	Cmd_R:			WORD;
	Cmd_CLen:		WORD;
	Cmd_RLen:		WORD;

	i : WORD;
	j : INT;


		(* per aggiornare la data e l'ora *)
	SetAnno: INT;
	SetMese: INT;
	SetGiorno: INT;
	SetOra: INT;
	SetMinuti: INT;
	SetSecondi: INT;

         (* specific for lux *)
	x: INT;
	NewValueTimer : DWORD;


	DummyWord: WORD;
	pioo: BOOL;
END_VAR
(*=== State machine ===*)
CASE Status OF
	0: (* Startup *)
		TxLen:=0; TxTrig:=FALSE;
		RxLen:=0;
		Enable:=TRUE;
		Status:=1;

	1: (* Wait incoming connection *)
		IF Connected THEN
			(* Log access *)
			LogEv(EL_Log,EO_VPN,1,5,'Remote');
			(* Send welcome message *)
			(*ADDSTRING(pTxData:=ADR(TxData), pString:=ADR(Remote_WELCOME), TxLen:=TxLen);
			TxTrig:=TRUE;*)
			Cmd_BufLen:=0;
			Cmd_St:=0;
			Status:=2;
		END_IF
		IF Error>1 THEN
			Enable:=FALSE;
			Status:=0;
		END_IF

	2: (* Wait command *)
		IF RxLen>0 THEN
			(*=== Interpreter start ===*)
			IF Cmd_BufLen+(RxLen/2)>=MAX_RECEIVE_TCP_SERVER THEN
				(* ERROR *)
				Cmd_BufLen:=0;
			ELSE
				i:=HEXTORAW(pString:=ADR(RxData), StringLen:=DINT_TO_WORD(RxLen), pData:=ADR(Cmd_Buf[Cmd_BufLen]));
				Cmd_BufLen:=Cmd_BufLen+i;
			END_IF
			IF Cmd_BufLen>=8 THEN
				Cmd_Buf_U16:=ADR(Cmd_Buf[6]);
				IF Cmd_BufLen>=(8+Cmd_Buf_U16^) THEN
					Cmd_CLen:=Cmd_Buf_U16^;
					Cmd_Buf_U16:=ADR(Cmd_Buf[0]); Cmd_Obj:=Cmd_Buf_U16^;
					Cmd_Buf_U16:=ADR(Cmd_Buf[2]); Cmd_ObjIdx:=Cmd_Buf_U16^;
					Cmd_Buf_U16:=ADR(Cmd_Buf[4]); Cmd_C:=Cmd_Buf_U16^;
					Command();
					Cmd_BufLen:=0;
				END_IF
			END_IF
			(*=== Interpreter end ===*)
			RxLen:=0;
		END_IF
		IF NOT Connected THEN
			Status:=0;
		END_IF

ELSE
	Status:=0;
END_CASE


(*=== Execute server lib ===*)
s1(
	xEnable				:= Enable,
	wPortNumber			:= Remote_PORT,
	tServerTimeOut		:= t#15m,
	ptSendData			:= ADR(TxData),
	diSendCount			:= TxLen,
	xStartSend			:= TxTrig,
	aReceiveBuffer		:= RxData,
	diReceiveCount		:= RxLen,
	xClientConnected	=> Connected,
	diError				=> Error
);
END_PROGRAM
ACTION Cmd_CRON:
(* Check index *)
IF Cmd_ObjIdx<1 OR Cmd_ObjIdx>11 THEN
	Cmd_R:=2;
	RETURN;
END_IF

(* Process command *)
CASE Cmd_C OF

	1: (* GET PROFILE *)
		IF Cmd_CLen<>3 THEN
			Cmd_R:=4;
		ELSE
			(* Load profile *)
			CronEd.CN_Sel:=WORD_TO_BYTE(Cmd_ObjIdx);
			Cmd_Buf_U16:=ADR(Cmd_Buf[8]);
			CronEd.CN_YSel:=Cmd_Buf_U16^;
			IF Cmd_Buf[10]<=10 THEN
				CronEd.PR_Sel:=Cmd_Buf[10];
				CronEd.PR_Load_Exe();
				(* Response data *)
				Cmd_RLen:=192;
				TxLen:=TxLen+RAWTOHEX(ADR(CronEd.PR.Setpoint),192,ADR(TxData[TxLen]));
			ELSE
				Cmd_R:=6;
			END_IF
		END_IF

	2: (* SET PROFILE *)
		IF Cmd_CLen<>(3+192) THEN
			Cmd_R:=4;
		ELSE
			(* Save profile *)
			CronEd.CN_Sel:=WORD_TO_BYTE(Cmd_ObjIdx);
			Cmd_Buf_U16:=ADR(Cmd_Buf[8]);
			CronEd.CN_YSel:=Cmd_Buf_U16^;
			IF Cmd_Buf[10]<=10 THEN
				CronEd.PR_Sel:=Cmd_Buf[10];
				MEMCPY(ADR(Cmd_Buf[11]),ADR(CronEd.PR.Setpoint),192);
				CronEd.PR_Save_Exe_Multi(); (* updated by DB - for saving profiles in eventually existing multiple crono files *)
			ELSE
				Cmd_R:=6;
			END_IF
		END_IF

	5: (* GET CALENDAR MONTH *)
		IF Cmd_CLen<>3 THEN
			Cmd_R:=4;
		ELSE
			(* Load calendar *)
			CronEd.CN_Sel:=WORD_TO_BYTE(Cmd_ObjIdx);
			Cmd_Buf_U16:=ADR(Cmd_Buf[8]);
			CronEd.CN_YSel:=Cmd_Buf_U16^;
			IF Cmd_Buf[10]>=1 AND Cmd_Buf[10]<=12 THEN
				CronEd.CA_Sel:=Cmd_Buf[10];
				CronEd.CA_Load_Exe();
				(* Response data *)
				Cmd_RLen:=32;
				TxLen:=TxLen+RAWTOHEX(ADR(CronEd.CA.Profile),32,ADR(TxData[TxLen]));
			ELSE
				Cmd_R:=6;
			END_IF
		END_IF

	6: (* SET CALENDAR MONTH *)
		IF Cmd_CLen<>(3+32) THEN
			Cmd_R:=4;
		ELSE
			(* Save calendar *)
			CronEd.CN_Sel:=WORD_TO_BYTE(Cmd_ObjIdx);
			Cmd_Buf_U16:=ADR(Cmd_Buf[8]);
			CronEd.CN_YSel:=Cmd_Buf_U16^;
			IF Cmd_Buf[10]>=1 AND Cmd_Buf[10]<=12 THEN
				CronEd.CA_Sel:=Cmd_Buf[10];
				MEMCPY(ADR(Cmd_Buf[11]),ADR(CronEd.CA.Profile),32);
				CronEd.CA_Save_Exe();
			ELSE
				Cmd_R:=6;
			END_IF
		END_IF

	9: (* CRON RESTART *)
		CASE Cmd_ObjIdx OF
			1: CRON01.InitOK:=FALSE;
			2: CRON02.InitOK:=FALSE;
			3: CRON03.InitOK:=FALSE;
			4: CRON04.InitOK:=FALSE;
			5: CRON05.InitOK:=FALSE;
			6: CRON06.InitOK:=FALSE;
			7: CRON07.InitOK:=FALSE;
			8: CRON08.InitOK:=FALSE;
			9: CRON09.InitOK:=FALSE;
			10: CRON10.InitOK:=FALSE;

		END_CASE

	10: (* SET Isteresi  *)
		CASE Cmd_ObjIdx OF

			1:	Cmd_Buf_U16:=ADR(Cmd_Buf[8]);
				CRON01.Histeresys := Cmd_Buf_U16^; 			(* Isteresi*)
			2:	Cmd_Buf_U16:=ADR(Cmd_Buf[8]);
				CRON02.Histeresys := Cmd_Buf_U16^; 			(* Isteresi*)
			3:	Cmd_Buf_U16:=ADR(Cmd_Buf[8]);
				CRON03.Histeresys := Cmd_Buf_U16^; 			(* Isteresi*)
			4:	Cmd_Buf_U16:=ADR(Cmd_Buf[8]);
				CRON04.Histeresys := Cmd_Buf_U16^; 			(* Isteresi*)
			5:	Cmd_Buf_U16:=ADR(Cmd_Buf[8]);
				CRON05.Histeresys := Cmd_Buf_U16^; 			(* Isteresi*)
			6:	Cmd_Buf_U16:=ADR(Cmd_Buf[8]);
				CRON06.Histeresys := Cmd_Buf_U16^; 			(* Isteresi*)
			7:	Cmd_Buf_U16:=ADR(Cmd_Buf[8]);
				CRON07.Histeresys := Cmd_Buf_U16^; 			(* Isteresi*)
			8:	Cmd_Buf_U16:=ADR(Cmd_Buf[8]);
				CRON08.Histeresys := Cmd_Buf_U16^; 			(* Isteresi*)
			9:	Cmd_Buf_U16:=ADR(Cmd_Buf[8]);
				CRON09.Histeresys := Cmd_Buf_U16^; 			(* Isteresi*)
			10:	Cmd_Buf_U16:=ADR(Cmd_Buf[8]);
				CRON10.Histeresys := Cmd_Buf_U16^; 			(* Isteresi*)

		END_CASE

	11: (* GET isteresi *)
		Cmd_RLen:=2;
		CASE Cmd_ObjIdx OF


			1: j:=(CRON01.Histeresys);
				TxLen:=TxLen+RAWTOHEX(ADR(j),2,ADR(TxData[TxLen]));
			2: j:=(CRON02.Histeresys);
				TxLen:=TxLen+RAWTOHEX(ADR(j),2,ADR(TxData[TxLen]));
			3: j:=(CRON03.Histeresys);
				TxLen:=TxLen+RAWTOHEX(ADR(j),2,ADR(TxData[TxLen]));
			4: j:=(CRON04.Histeresys);
				TxLen:=TxLen+RAWTOHEX(ADR(j),2,ADR(TxData[TxLen]));
			5: j:=(CRON05.Histeresys);
				TxLen:=TxLen+RAWTOHEX(ADR(j),2,ADR(TxData[TxLen]));
			6: j:=(CRON06.Histeresys);
				TxLen:=TxLen+RAWTOHEX(ADR(j),2,ADR(TxData[TxLen]));
			7: j:=(CRON07.Histeresys);
				TxLen:=TxLen+RAWTOHEX(ADR(j),2,ADR(TxData[TxLen]));
			8: j:=(CRON08.Histeresys);
				TxLen:=TxLen+RAWTOHEX(ADR(j),2,ADR(TxData[TxLen]));
			9: j:=(CRON09.Histeresys);
				TxLen:=TxLen+RAWTOHEX(ADR(j),2,ADR(TxData[TxLen]));
			10: j:=(CRON10.Histeresys);
				TxLen:=TxLen+RAWTOHEX(ADR(j),2,ADR(TxData[TxLen]));

		END_CASE
ELSE
	Cmd_R:=3;
END_CASE
END_ACTION
ACTION cmd_LUX:
(* Check index *)
IF Cmd_ObjIdx < 1 OR Cmd_ObjIdx > MAX_LuxElement THEN
	Cmd_R := 2; (* //id del lux fuori range*)
	RETURN ;
END_IF
(*
x := 1 ;
WHILE ( Cmd_ObjIdx <> TabDefaultLux [ x ] . LuxNumber ) AND ( x <=MAX_LUXNUM ) DO
	x := x + 1 ;
END_WHILE

IF Cmd_ObjIdx = TabDefaultLux [ x ] . LuxNumber THEN
*)
	(* Process command *)
 	CASE Cmd_C OF

		0 : (* Restore default functioning mode *)
		CASE Cmd_ObjIdx OF

			1:	LuxElement01.CTRL_MODE	:= 2;
			2:	LuxElement02.CTRL_MODE	:= 2;
			3:	LuxElement03.CTRL_MODE	:= 2;
			4:	LuxElement04.CTRL_MODE	:= 2;
			5:	LuxElement05.CTRL_MODE	:= 2;
			6:	LuxElement06.CTRL_MODE	:= 2;
			7:	LuxElement07.CTRL_MODE	:= 2;
			8:	LuxElement08.CTRL_MODE	:= 2;
			9:	LuxElement09.CTRL_MODE	:= 2;
			10:	LuxElement10.CTRL_MODE	:= 2;
			11:	LuxElement11.CTRL_MODE	:= 2;
			12:	LuxElement12.CTRL_MODE	:= 2;
		END_CASE		(*	LuxElement [ x ] . CTRL_MODE := LuxElement [ x ] . CTRL_MODE_backUp ;
			LuxElement [ x ] (     WORKINGTIME := WORKINGTIME_n [ x ] ,
							POWERONCYCLES :=
							POWERONCYCLES_n [ x ] ,
							ENERGYCOUNTER := ENERGYCOUNTER_n [ x ] ,
							ENERGYCOUNTER_T :=
							ENERGYCOUNTER_T_n [ x ] ,
							CtrlExton := KEYON ) ;*)

		1 : (* Reset statistic counter *)

		pioo:=0;

		(*	LuxElement [ x ] . StatReset (  WORKINGTIME := WORKINGTIME_n [ x ] ,
									POWERONCYCLES := POWERONCYCLES_n [ x ] ,
									ENERGYCOUNTER :=ENERGYCOUNTER_n [ x ] ,
									ENERGYCOUNTER_T:= ENERGYCOUNTER_T_n [ x ] ,
									CtrlExton :=KEYON ) ;*)

		2:(* Switch On (command=2)  *)

		CASE Cmd_ObjIdx OF

			1:	LuxElement01.CTRL_MODE	:= 1;
			2:	LuxElement02.CTRL_MODE	:= 1;
			3:	LuxElement03.CTRL_MODE	:= 1;
			4:	LuxElement04.CTRL_MODE	:= 1;
			5:	LuxElement05.CTRL_MODE	:= 1;
			6:	LuxElement06.CTRL_MODE	:= 1;
			7:	LuxElement07.CTRL_MODE	:= 1;
			8:	LuxElement08.CTRL_MODE	:= 1;
			9:	LuxElement09.CTRL_MODE	:= 1;
			10:	LuxElement10.CTRL_MODE	:= 1;
			11:	LuxElement11.CTRL_MODE	:= 1;
			12:	LuxElement12.CTRL_MODE	:= 1;
		END_CASE




		 3 : (*  Off (command=3) lux *)
		CASE Cmd_ObjIdx OF

			1:	LuxElement01.CTRL_MODE	:= 0;
			2:	LuxElement02.CTRL_MODE	:= 0;
			3:	LuxElement03.CTRL_MODE	:= 0;
			4:	LuxElement04.CTRL_MODE	:= 0;
			5:	LuxElement05.CTRL_MODE	:= 0;
			6:	LuxElement06.CTRL_MODE	:= 0;
			7:	LuxElement07.CTRL_MODE	:= 0;
			8:	LuxElement08.CTRL_MODE	:= 0;
			9:	LuxElement09.CTRL_MODE	:= 0;
			10:	LuxElement10.CTRL_MODE	:= 0;
			11:	LuxElement11.CTRL_MODE	:= 0;
			12:	LuxElement12.CTRL_MODE	:= 0;
		END_CASE




		(*	CASE Cmd_C OF
				2 : (*switch a Manuale ON*)
					LuxElement [ x ] . CTRL_MODE := 1 ; (*// Set to manuale ON *)
					LuxElement [ x ] (     WORKINGTIME := WORKINGTIME_n [ x ] ,
									POWERONCYCLES:= POWERONCYCLES_n [ x ] ,
									ENERGYCOUNTER :=ENERGYCOUNTER_n [ x ] ,
									ENERGYCOUNTER_T :=ENERGYCOUNTER_T_n [ x ] ,
									CtrlExton := KEYON ) ;

				3 : (*switch a Manuale OFF*)
					(*LuxElement [ x ] . CTRL_MODE := 0 ; (*// Set to manuale OFF *)
					LuxElement [ x ] (     WORKINGTIME := WORKINGTIME_n [ x ] ,
									POWERONCYCLES:= POWERONCYCLES_n [ x ] ,
									ENERGYCOUNTER :=ENERGYCOUNTER_n [ x ] ,
									ENERGYCOUNTER_T :=ENERGYCOUNTER_T_n [ x ] ,
									CtrlExton := KEYON ) ;*)

			END_CASE*)

		4 : (* Modify timer value *)
		pioo:=0;
		(*	IF TabDefaultLux [ x ] . Mode = 03 THEN
				(*la modifica ha senso per i lux a timer*)
				NewValueTimer := BYTE_TO_DWORD ( Cmd_Buf [ 8 ] ) ;
				NewValueTimer := SHL ( NewValueTimer , 8 ) ;	
				NewValueTimer := NewValueTimer + BYTE_TO_DWORD ( Cmd_Buf [ 9 ] ) ;
				NewValueTimer := SHL ( NewValueTimer , 8 ) ;
				NewValueTimer := NewValueTimer + BYTE_TO_DWORD ( Cmd_Buf [ 10 ] ) ;
				NewValueTimer := SHL ( NewValueTimer , 8 ) ;
				NewValueTimer := NewValueTimer + BYTE_TO_DWORD ( Cmd_Buf [ 11 ] ) ;
				(*TabLuxPsg [ x ] . TimerOn := DWORD_TO_TIME ( NewValueTimer *1000 ) ;*) (*REMOVE THIS LINE *)

				FOR x := 1 TO MAX_LUXNUM DO
					IF LuxElement [ x ] . ID = Cmd_ObjIdx THEN
						LuxElement [ x ] . LuxTimer := DWORD_TO_TIME (NewValueTimer * 1000 ) ; (*//set del nuovo valore del timer del lux*)
					END_IF
				END_FOR
			ELSE
				Cmd_R := 3 ; (*//Comando errato / non previsto*)
			END_IF
		(* 5: (* Modify dimming value for timer control *) *)
		(* 6: (* Modify dimming value for key control *) *)

		(* 7: (* Modify start and stop orari di funzionamento dei lux a timer *) *) *)
		ELSE
			Cmd_R := 3 ; (*//Comando errato / non previsto*)
		END_CASE

(*
ELSE
	Cmd_R := 2 ; (*//id del lux non presente in lista*)
END_IF
*)
END_ACTION
ACTION Cmd_SYS:
(* Check index *)
IF Cmd_ObjIdx<>0 THEN
	Cmd_R:=2;
	RETURN;
END_IF

(* Process command *)
CASE Cmd_C OF

	0: (* ECHO *)
		IF Cmd_CLen<>0 THEN
			TxLen:=0;
		END_IF

	1: (* LOG REQUEST *)
		(*LogTrig(); *)
		PLC_PRG.RichiestaDaRemoto:=TRUE;


	2: (* REARM *)
		Sys.Warning:=FALSE;
		Sys.Alarm:=FALSE;
		Sys.AlarmStop:=FALSE;

	3: (* GET INFO1 *)
		Cmd_RLen:=6;
		TxLen:=TxLen+RAWTOHEX(ADR(Plant_SN),4,ADR(TxData[TxLen]));
		TxLen:=TxLen+RAWTOHEX(ADR(Plant_SW_VER),2,ADR(TxData[TxLen]));


(*	4: (*  Scrivo i Parametri gestione Impianto   *)

			Cmd_Buf_U16:=ADR(Cmd_Buf[8]);
			DelayAllarmeTemperaturaNonRaggiunta := Cmd_Buf_U16^; 			(* Ritardo Allarme dall'avvio Caldaia*)
			Cmd_Buf_U16:=ADR(Cmd_Buf[10]);
			DeltaInterventoAllarmeTempeaturaNonRaggiuta := Cmd_Buf_U16^;	(* Delta Soglia Temperatura per Allarme Temperatura Non Raggiunta *)
			Cmd_Buf_U16:=ADR(Cmd_Buf[12]);
			OffsetSetPointManuale := Cmd_Buf_U16^; 							(* Offest Perdite Scambiatore 1  *)
			Cmd_Buf_U16:=ADR(Cmd_Buf[14]);
			OffsetSetPointManuale2 := Cmd_Buf_U16^; 						(* Offest Perdite Scambiatore 1  *)
			Cmd_Buf_U16:=ADR(Cmd_Buf[12]);
			BitAbilitaBoost :=INT_TO_BOOL( Cmd_Buf_U16^); 					(* Abilitazione controllo Boost  *)
			Cmd_Buf_U16:=ADR(Cmd_Buf[14]);
			RifOffsetBoost := Cmd_Buf_U16^; 								(* Offset al Setpoint della Caldaia per azione di Boost  *)


	5: (*  Leggi i parametri gestione Impianto  *)

			Cmd_RLen:=18;
			j:=(DelayAllarmeTemperaturaNonRaggiunta);   				(* Ritardo Allarme dall'avvio Caldaia*)
			TxLen:=TxLen+RAWTOHEX(ADR(j),2,ADR(TxData[TxLen]));
			j:=(DeltaInterventoAllarmeTempeaturaNonRaggiuta);			(* Delta Soglia Temperatura per Allarme Temperatura Non Raggiunta *)
			TxLen:=TxLen+RAWTOHEX(ADR(j),2,ADR(TxData[TxLen]));
			j:=(OffsetSetPointManuale);									(* Offest Perdite Scambiatore 1  *)
			TxLen:=TxLen+RAWTOHEX(ADR(j),2,ADR(TxData[TxLen]));
			j:=(OffsetSetPointManuale2);								(* Offest Perdite Scambiatore 2  *)
			TxLen:=TxLen+RAWTOHEX(ADR(j),2,ADR(TxData[TxLen]));
			j:=BOOL_TO_INT(BitAbilitaBoost);							(* Abilitazione controllo Boost  *)
			TxLen:=TxLen+RAWTOHEX(ADR(j),2,ADR(TxData[TxLen]));
			j:=BOOL_TO_INT(BitAbilitaBoost);										(* Offset al Setpoint della Caldaia per azione di Boost   *)
			TxLen:=TxLen+RAWTOHEX(ADR(j),2,ADR(TxData[TxLen]));




	6: (*  Scrivo i Parametri gestione Impianto - Antigelo   *)

			Cmd_Buf_U16:=ADR(Cmd_Buf[8]);
			SogliaMinStartAntigelo := Cmd_Buf_U16^; 			(* Soglia mininma Start Antigelo *)
			Cmd_Buf_U16:=ADR(Cmd_Buf[10]);
			SogliaMinStopAntigelo := Cmd_Buf_U16^;				(* Soglia Massima Stop Antigelo *)
			Cmd_Buf_U16:=ADR(Cmd_Buf[12]);
			BitAbilitaAntigelo :=INT_TO_BOOL( Cmd_Buf_U16^); 	(* Abilitazione Antigelo  *)

	7: (*  Leggi i parametri gestione Impianto - Antigelo *)

			Cmd_RLen:=14;
			j:=(SogliaMinStartAntigelo); 							(* Soglia mininma Start Antigelo *)
			TxLen:=TxLen+RAWTOHEX(ADR(j),2,ADR(TxData[TxLen]));
			j:=(SogliaMinStopAntigelo);								(* Soglia Massima Stop Antigelo *)
			TxLen:=TxLen+RAWTOHEX(ADR(j),2,ADR(TxData[TxLen]));
			j:=BOOL_TO_INT(BitAbilitaAntigelo);						(* Abilitazione Antigelo  *)
			TxLen:=TxLen+RAWTOHEX(ADR(j),2,ADR(TxData[TxLen]));

(*	10: (*  Scrivo i Parametri per la gestione della velocità dei circolatori sui primari   *)

			Cmd_Buf_U16:=ADR(Cmd_Buf[8]);
			PercVelMin := Cmd_Buf_U16^;
			Cmd_Buf_U16:=ADR(Cmd_Buf[10]);
			PercVelMax := Cmd_Buf_U16^;
			Cmd_Buf_U16:=ADR(Cmd_Buf[12]);
			ErroreTempMax := Cmd_Buf_U16^;
			Cmd_Buf_U16:=ADR(Cmd_Buf[14]);
			ErroreTempMin := Cmd_Buf_U16^;

	11: (*  Leggo i Parametri per la gestione della velocità dei circolatori sui primari   *)

			Cmd_RLen:=8;
			j:=(PercVelMin);
			TxLen:=TxLen+RAWTOHEX(ADR(j),2,ADR(TxData[TxLen]));
			j:=(PercVelMax);
			TxLen:=TxLen+RAWTOHEX(ADR(j),2,ADR(TxData[TxLen]));
			j:=(ErroreTempMax);
			TxLen:=TxLen+RAWTOHEX(ADR(j),2,ADR(TxData[TxLen]));
			j:=(ErroreTempMin);
			TxLen:=TxLen+RAWTOHEX(ADR(j),2,ADR(TxData[TxLen]));


	12: (*  Scrivo i Parametri per la gestione della velocità dei circolatori sui primari   *)


				Cmd_Buf_U16:=ADR(Cmd_Buf[8]);
				CAS01.DeltaTempThr := Cmd_Buf_U16^;
				Cmd_Buf_U16:=ADR(Cmd_Buf[10]);
				CAS01.Tmonitor_Off := DWORD_TO_TIME((Cmd_Buf_U16^)*60*1000);
				Cmd_Buf_U16:=ADR(Cmd_Buf[12]);
				CAS01.Tmonitor_On := DWORD_TO_TIME((Cmd_Buf_U16^)*60*1000);

	13: (*  Leggo i Parametri per la gestione della velocità dei circolatori sui primari   *)


				Cmd_RLen:=6;
				j:=(CAS01.DeltaTempThr);
				TxLen:=TxLen+RAWTOHEX(ADR(j),2,ADR(TxData[TxLen]));
				j:=DWORD_TO_WORD(TIME_TO_DWORD((CAS01.Tmonitor_Off)/60/1000));
				TxLen:=TxLen+RAWTOHEX(ADR(j),2,ADR(TxData[TxLen]));
				j:=DWORD_TO_WORD(TIME_TO_DWORD((CAS01.Tmonitor_On)/60/1000));
				TxLen:=TxLen+RAWTOHEX(ADR(j),2,ADR(TxData[TxLen]));


*) *)


	14: (*  Imposto data e ora del PLC  *)


			Cmd_Buf_U16:=ADR(Cmd_Buf[8]);
			SetAnno:= Cmd_Buf_U16^; 												(* Anno *)
			Cmd_Buf_U16:=ADR(Cmd_Buf[10]);
			SetMese:= Cmd_Buf_U16^;												 	(* mese *)
			Cmd_Buf_U16:=ADR(Cmd_Buf[12]);
			SetGiorno:=( Cmd_Buf_U16^);											 	(* Giorno *)
			Cmd_Buf_U16:=ADR(Cmd_Buf[14]);
			SetOra:=( Cmd_Buf_U16^); 												(* ora *)
			Cmd_Buf_U16:=ADR(Cmd_Buf[16]);
			SetMinuti:= ( Cmd_Buf_U16^);										 	(* Minuti *)
			Cmd_Buf_U16:=ADR(Cmd_Buf[18]);
			SetSecondi:= ( Cmd_Buf_U16^);										 	(* secondi *)

	(*		SysRtcSetTime(SetDataTime(DWORD_TO_INT(ADR(Cmd_Buf[8])),				(* Anno *)
										DWORD_TO_INT(ADR(Cmd_Buf[10])),				(* mese *)
										DWORD_TO_INT(ADR(Cmd_Buf[11])),				(* Giorno *)
										DWORD_TO_INT(ADR(Cmd_Buf[12])),				(* ora *)
										DWORD_TO_INT(ADR(Cmd_Buf[13])),				(* Minuti *)
										DWORD_TO_INT(ADR(Cmd_Buf[14]))				(* secondi *)
										)); *)

		SysRtcSetTime((SetDataTime(SetAnno,SetMese,SetGiorno,SetOra,SetMinuti,SetSecondi)));


ELSE
	Cmd_R:=3;
END_CASE
END_ACTION
ACTION cmd_VAR:
(* Check index *)
IF Cmd_ObjIdx<1 OR  Cmd_ObjIdx>3   THEN
	Cmd_R:=2;
	RETURN;
END_IF

(* Process command *)

CASE Cmd_C OF

	1: (* SET Comandi  *)
		CASE Cmd_ObjIdx OF
			1:	Cmd_Buf_U16:=ADR(Cmd_Buf[8]);
				PLC_PRG.SogliaLux01 := (Cmd_Buf_U16^);     (* Val 01 *)
				Cmd_Buf_U16:=ADR(Cmd_Buf[10]);
				PLC_PRG.IsteresiLux01 :=(Cmd_Buf_U16^);	 (* Val 02 *)
				Cmd_Buf_U16:=ADR(Cmd_Buf[12]);
				PLC_PRG.SogliaLux02 := (Cmd_Buf_U16^);	 (* Val 03 *)
				Cmd_Buf_U16:=ADR(Cmd_Buf[14]);
				PLC_PRG.IsteresiLux02 := (Cmd_Buf_U16^);	 (* Val 04 *)
				Cmd_Buf_U16:=ADR(Cmd_Buf[16]);
				PLC_PRG.SogliaLux03 := (Cmd_Buf_U16^);	 	(* Val 05 *)
				Cmd_Buf_U16:=ADR(Cmd_Buf[18]);
				PLC_PRG.IsteresiLux03 := (Cmd_Buf_U16^);	 (* Val 06 *)
				Cmd_Buf_U16:=ADR(Cmd_Buf[20]);
				PLC_PRG.SogliaLux04 := (Cmd_Buf_U16^);			 (* Val 07 *)
				Cmd_Buf_U16:=ADR(Cmd_Buf[22]);
				PLC_PRG.IsteresiLux04 := (Cmd_Buf_U16^);	 		(* Val 08 *)
				Cmd_Buf_U16:=ADR(Cmd_Buf[24]);
				PLC_PRG.SogliaLux05 := (Cmd_Buf_U16^);	 		(* Val 09 *)
				Cmd_Buf_U16:=ADR(Cmd_Buf[26]);
				PLC_PRG.IsteresiLux05 := (Cmd_Buf_U16^);	 		(* Val 10 *)



			2:	Cmd_Buf_U16:=ADR(Cmd_Buf[8]);
				PLC_PRG.SogliaLux06 := (Cmd_Buf_U16^);     (* Val 01 *)
				Cmd_Buf_U16:=ADR(Cmd_Buf[10]);
				PLC_PRG.IsteresiLux06 :=(Cmd_Buf_U16^);	 (* Val 02 *)
				Cmd_Buf_U16:=ADR(Cmd_Buf[12]);
				PLC_PRG.SogliaLux07 := (Cmd_Buf_U16^);	 (* Val 03 *)
				Cmd_Buf_U16:=ADR(Cmd_Buf[14]);
				PLC_PRG.IsteresiLux07 := (Cmd_Buf_U16^);	 (* Val 04 *)
				Cmd_Buf_U16:=ADR(Cmd_Buf[16]);
				PLC_PRG.SogliaLux08 := (Cmd_Buf_U16^);	 	(* Val 05 *)
				Cmd_Buf_U16:=ADR(Cmd_Buf[18]);
				PLC_PRG.IsteresiLux08 := (Cmd_Buf_U16^);	 (* Val 06 *)
				Cmd_Buf_U16:=ADR(Cmd_Buf[20]);
				PLC_PRG.SogliaLux09 := (Cmd_Buf_U16^);			 (* Val 07 *)
				Cmd_Buf_U16:=ADR(Cmd_Buf[22]);
				PLC_PRG.IsteresiLux09 := (Cmd_Buf_U16^);	 		(* Val 08 *)
				Cmd_Buf_U16:=ADR(Cmd_Buf[24]);
				PLC_PRG.SogliaLux10 := (Cmd_Buf_U16^);	 		(* Val 09 *)
				Cmd_Buf_U16:=ADR(Cmd_Buf[26]);
				PLC_PRG.IsteresiLux10 := (Cmd_Buf_U16^);	 		(* Val 10 *)

			3:	Cmd_Buf_U16:=ADR(Cmd_Buf[8]);
				PLC_PRG.SogliaLux11 := (Cmd_Buf_U16^);     (* Val 01 *)
				Cmd_Buf_U16:=ADR(Cmd_Buf[10]);
				PLC_PRG.IsteresiLux11 :=(Cmd_Buf_U16^);	 (* Val 02 *)
				Cmd_Buf_U16:=ADR(Cmd_Buf[12]);
				PLC_PRG.SogliaLux12 := (Cmd_Buf_U16^);	 (* Val 03 *)
				Cmd_Buf_U16:=ADR(Cmd_Buf[14]);
				PLC_PRG.IsteresiLux12 := (Cmd_Buf_U16^);	 (* Val 04 *)
				Cmd_Buf_U16:=ADR(Cmd_Buf[16]);
				PLC_PRG.delayOffLux:= (Cmd_Buf_U16^);	 	(* Val 05 *)
				Cmd_Buf_U16:=ADR(Cmd_Buf[18]);
				DummyWord := (Cmd_Buf_U16^);	 (* Val 06 *)
				Cmd_Buf_U16:=ADR(Cmd_Buf[20]);
				DummyWord := (Cmd_Buf_U16^);			 (* Val 07 *)
				Cmd_Buf_U16:=ADR(Cmd_Buf[22]);
				DummyWord := (Cmd_Buf_U16^);	 		(* Val 08 *)
				Cmd_Buf_U16:=ADR(Cmd_Buf[24]);
				DummyWord := (Cmd_Buf_U16^);	 		(* Val 09 *)
				Cmd_Buf_U16:=ADR(Cmd_Buf[26]);
				DummyWord := (Cmd_Buf_U16^);	 		(* Val 10 *)




		END_CASE


	2: (* GET Comandi  *)
		CASE Cmd_ObjIdx OF

			1: (*  Leggi i parametri gestione Impianto  *)
			Cmd_RLen:=10;
			j:=(PLC_PRG.SogliaLux01);
			TxLen:=TxLen+RAWTOHEX(ADR(j),2,ADR(TxData[TxLen]));
			j:=(PLC_PRG.IsteresiLux01);
			TxLen:=TxLen+RAWTOHEX(ADR(j),2,ADR(TxData[TxLen]));
			j:=(PLC_PRG.SogliaLux02);
			TxLen:=TxLen+RAWTOHEX(ADR(j),2,ADR(TxData[TxLen]));
			j:=(PLC_PRG.IsteresiLux02);
			TxLen:=TxLen+RAWTOHEX(ADR(j),2,ADR(TxData[TxLen]));
			j:=(PLC_PRG.SogliaLux03);
			TxLen:=TxLen+RAWTOHEX(ADR(j),2,ADR(TxData[TxLen]));
			j:=(PLC_PRG.IsteresiLux03);
			TxLen:=TxLen+RAWTOHEX(ADR(j),2,ADR(TxData[TxLen]));
			j:=(PLC_PRG.SogliaLux04);
			TxLen:=TxLen+RAWTOHEX(ADR(j),2,ADR(TxData[TxLen]));
			j:=(PLC_PRG.IsteresiLux04);
			TxLen:=TxLen+RAWTOHEX(ADR(j),2,ADR(TxData[TxLen]));
			j:=(PLC_PRG.SogliaLux05);
			TxLen:=TxLen+RAWTOHEX(ADR(j),2,ADR(TxData[TxLen]));
			j:=(PLC_PRG.IsteresiLux05);
			TxLen:=TxLen+RAWTOHEX(ADR(j),2,ADR(TxData[TxLen]));

			2: (*  Leggi i parametri gestione Impianto  *)
			Cmd_RLen:=10;
			j:=(PLC_PRG.SogliaLux06);
			TxLen:=TxLen+RAWTOHEX(ADR(j),2,ADR(TxData[TxLen]));
			j:=(PLC_PRG.IsteresiLux06);
			TxLen:=TxLen+RAWTOHEX(ADR(j),2,ADR(TxData[TxLen]));
			j:=(PLC_PRG.SogliaLux07);
			TxLen:=TxLen+RAWTOHEX(ADR(j),2,ADR(TxData[TxLen]));
			j:=(PLC_PRG.IsteresiLux07);
			TxLen:=TxLen+RAWTOHEX(ADR(j),2,ADR(TxData[TxLen]));
			j:=(PLC_PRG.SogliaLux08);
			TxLen:=TxLen+RAWTOHEX(ADR(j),2,ADR(TxData[TxLen]));
			j:=(PLC_PRG.IsteresiLux08);
			TxLen:=TxLen+RAWTOHEX(ADR(j),2,ADR(TxData[TxLen]));
			j:=(PLC_PRG.SogliaLux09);
			TxLen:=TxLen+RAWTOHEX(ADR(j),2,ADR(TxData[TxLen]));
			j:=(PLC_PRG.IsteresiLux09);
			TxLen:=TxLen+RAWTOHEX(ADR(j),2,ADR(TxData[TxLen]));
			j:=(PLC_PRG.SogliaLux10);
			TxLen:=TxLen+RAWTOHEX(ADR(j),2,ADR(TxData[TxLen]));
			j:=(PLC_PRG.IsteresiLux10);
			TxLen:=TxLen+RAWTOHEX(ADR(j),2,ADR(TxData[TxLen]));

			3: (*  Leggi i parametri gestione Impianto  *)
			Cmd_RLen:=10;
			j:=(PLC_PRG.SogliaLux11);
			TxLen:=TxLen+RAWTOHEX(ADR(j),2,ADR(TxData[TxLen]));
			j:=(PLC_PRG.IsteresiLux11);
			TxLen:=TxLen+RAWTOHEX(ADR(j),2,ADR(TxData[TxLen]));
			j:=(PLC_PRG.SogliaLux12);
			TxLen:=TxLen+RAWTOHEX(ADR(j),2,ADR(TxData[TxLen]));
			j:=(PLC_PRG.IsteresiLux12);
			TxLen:=TxLen+RAWTOHEX(ADR(j),2,ADR(TxData[TxLen]));
			j:=(PLC_PRG.delayOffLux);
			TxLen:=TxLen+RAWTOHEX(ADR(j),2,ADR(TxData[TxLen]));
			j:=(0);
			TxLen:=TxLen+RAWTOHEX(ADR(j),2,ADR(TxData[TxLen]));
			j:=(0);
			TxLen:=TxLen+RAWTOHEX(ADR(j),2,ADR(TxData[TxLen]));
			j:=(0);
			TxLen:=TxLen+RAWTOHEX(ADR(j),2,ADR(TxData[TxLen]));
			j:=(0);
			TxLen:=TxLen+RAWTOHEX(ADR(j),2,ADR(TxData[TxLen]));
			j:=(0);
			TxLen:=TxLen+RAWTOHEX(ADR(j),2,ADR(TxData[TxLen]));





		END_CASE

ELSE
	Cmd_R:=3;
END_CASE
END_ACTION
ACTION Command:
(* Default response OK/NODATA *)
Cmd_R:=0;
Cmd_RLen:=0;
TxLen:=16;

(* Check object *)
CASE Cmd_Obj OF

	EO_SYS:
		Cmd_SYS();

	EO_LUX:
		Cmd_LUX();

	EO_CRON,EO_THER:
		Cmd_CRON();

	EO_VAR:
		Cmd_VAR();



ELSE
	Cmd_R:=1;
END_CASE

(* Generate response *)
IF TxLen>0 THEN
	RAWTOHEX(ADR(Cmd_Obj)	,2,ADR(TxData[ 0]));
	RAWTOHEX(ADR(Cmd_ObjIdx),2,ADR(TxData[ 4]));
	RAWTOHEX(ADR(Cmd_R)		,2,ADR(TxData[ 8]));
	RAWTOHEX(ADR(Cmd_RLen)	,2,ADR(TxData[12]));
	TxTrig:=TRUE;
END_IF
END_ACTION

(* POU Utils Functions/TCPSERVER, ST *)
FUNCTION_BLOCK TCPSERVER
(***********************************************************************************************************	*)
(* Version: 1.6                                    			          											*)
(* Date: 11.02.2011                                   					          							    *)
(***********************************************************************************************************	*)
(* WAGO Kontakttechnik GmbH Hansastr. 27 32423 Minden(Westf.)													*)
(* Tel. +0049 571/887-0 Fax. +0049 571/887-0																	*)
(* Author: VB																									*)
(***********************************************************************************************************	*)
(*Description:	A TCP server to read and write data													       		*)
(*Historie:																										*)
(*Version 1.6: 11.02.2011: Changes according to 750-880/881											 			*)
(*Version 1.5: 27.11.2008 Bugfix allow reuse port																*)
(*Version 1.4: 13.10.2008 Bugfix transmitting large data														*)
(*Version 1.3: 15.01.2007 Changes according to FW11																*)
(*Version 1.2: 09.03.2006 Changes for socket handle 0											       			*)
(*Version 1.1: 14.02.2005 Release																				*)
(***********************************************************************************************************	*)
VAR CONSTANT
	STATE_INIT     				 : BYTE:= 0;
	STATE_OPEN     				 : BYTE:= 1;
	STATE_TX       				 : BYTE:= 20;
	STATE_RX       				 : BYTE:= 30;
	STATE_CLOSE    				 : BYTE:= 40;
	STATE_ERROR_TRAP		 	 : BYTE:= 200;
END_VAR
VAR_INPUT
	xEnable    					: BOOL;	 (* Set TRUE to enable function block *)
	wPortNumber					: WORD;  (* Port *)
	tServerTimeOut				: TIME:=t#50s;
	ptSendData					: POINTER TO ARRAY[0..MAX_SEND_TCP_SERVER] OF BYTE;
	diSendCount					: DINT;
END_VAR
VAR_OUTPUT
	xClientConnected  			: BOOL:= FALSE;
	diError 					: DINT:= 0;
END_VAR
(* Status Codes -----------------------------------------
	16#8001 => No socket descriptor available 
	16#8002 => SysSockBind fails 
	16#8003 => SysSockListen fails 
	16#8004 => switching to none blocking mode fails
	16#8005 => SysSockClose() returns FALSE 
    16#8006 => SysSockConnect() fails
    16#8007 => SysSockSend() fails
	16#8008 => error state machine 
	16#8009 => timeout while waiting for data from server 
	16#0001 => server waiting for client to establish connection
------------------------------------------------------------*)
VAR_IN_OUT
	xStartSend					: BOOL;
	aReceiveBuffer				: ARRAY [0..MAX_RECEIVE_TCP_SERVER] OF BYTE;
	diReceiveCount				: DINT;
END_VAR

VAR
	m_State    					: BYTE:= 0;
	m_ReceiveBuffer				: ARRAY [0..MAX_RECEIVE_TCP_SERVER_SOCKET] OF BYTE;
	m_ServerSocket				: DINT:= SOCKET_INVALID;
	m_Socket					: DINT:= SOCKET_INVALID;
	m_AddressInfo				: SOCKADDRESS;
	m_BytesReceived				: DINT;
	m_diReturn					: DINT;
	m_xReturn					: BOOL;
	m_SizeSockadr				: DWORD;
	m_ConnectionWatchdog		: TON;
	m_Flags						: DINT;
	m_NoneBlocking   			: DINT:= 1;
	m_Blocking   				: DINT:= 0;
	i							: INT;
	m_count						: DINT;
	diOption					: DINT := 1;
	on: DINT;
END_VAR
IF xEnable THEN
	CASE m_State OF
		STATE_INIT:
			(* Create Socket *)
			m_ServerSocket:= SysSockCreate( SOCKET_AF_INET, SOCKET_STREAM, 0);
			IF m_ServerSocket = SOCKET_INVALID THEN
				(* *)
				diError:= 16#8001;
				m_State:= STATE_ERROR_TRAP;
				RETURN;
			ELSE
				;
			END_IF
			(* Address bindings *)
			(********************)
			on:=1;
			SysSockSetOption( m_ServerSocket, SOCKET_SOL, SOCKET_SO_REUSEADDR, ADR(on), SIZEOF(on) );

			m_AddressInfo.sin_family:= SOCKET_AF_INET;
			m_AddressInfo.sin_port  := SysSockHtons( wPortNumber);
			m_AddressInfo.sin_addr  := SOCKET_INADDR_ANY;
			IF NOT SysSockBind( m_ServerSocket, ADR(m_AddressInfo), SIZEOF(m_AddressInfo)) THEN
				diError:= 16#8002;
				m_State:= STATE_ERROR_TRAP;
				RETURN;
			END_IF
			(* Wait for connections *)
			(************************)
			IF NOT SysSockListen( m_ServerSocket, 1) THEN
				diError:= 16#8003;
				m_State:= STATE_ERROR_TRAP;
			END_IF

			(* Puts SOCKET in NonBlocking mode *)
			m_diReturn:= SysSockIoctl( m_ServerSocket, SOCKET_FIONBIO, ADR(m_NoneBlocking));

			m_State:= STATE_OPEN;


		STATE_OPEN: 	(* Waiting for incomming connection *)
				m_SizeSockadr:=SIZEOF(m_AddressInfo);
				m_Socket:= SysSockAccept( m_ServerSocket, ADR(m_AddressInfo), ADR(m_SizeSockadr));
				diError:=State_open;
				IF m_Socket <> SOCKET_INVALID THEN
					xClientConnected:=TRUE;
					(*Set Push-Bit:new V1.5*)
					IF ADR(%MW0)=16#30000000  OR ADR(%MW0)=16#20000000 THEN (*841 or 881*)
						SysSockSetOption(
							diSocket:=m_Socket,
							diLevel:=6,
							diOption:=SOCKET_TCP_NODELAY,
							pOptionValue:=ADR(diOption),
							diOptionLength:=SIZEOF(diOption));
					ELSE
							;
					END_IF
					SysSockIoctl( m_Socket, SOCKET_FIONBIO, ADR(m_NoneBlocking));
					m_State:= STATE_RX;
					diError:=0;
				END_IF

		STATE_RX:
					m_BytesReceived:= SysSockRecv( m_Socket, ADR(m_ReceiveBuffer), SIZEOF(m_ReceiveBuffer), 0);
					CASE m_BytesReceived OF
					-1:(*no data available or error occured*)
						m_ConnectionWatchdog(IN:=TRUE , PT:=tServerTimeOut );
						IF m_connectionWatchdog.Q THEN
							m_State:= STATE_CLOSE;
							m_ConnectionWatchdog(IN:=FALSE);(*reset connection watchdog*)
							diError := 16#8009;
						END_IF
					0:(* socket was "gracefully closed"  *)
						m_State:= STATE_CLOSE;
						diError := 16#8003;
					ELSE
						(* Copy received data into receive buffer *)
						(********************************)
						FOR i:= 0 TO DINT_TO_INT(m_BytesReceived	)-1 DO
							aReceiveBuffer[diReceiveCount]:= m_ReceiveBuffer[i];
							diReceiveCount:=(diReceiveCount+1) MOD SIZEOF(aReceiveBuffer);
						END_FOR

						m_ConnectionWatchdog(IN:=FALSE);(*reset connection watchdog*)
					END_CASE

				(*send data*)
				IF xStartSend	 THEN
					m_State := STATE_TX;
				END_IF

	STATE_TX:	 (* send TCP-message *)
		m_diReturn := SysSockSend(diSocket := m_Socket,
								  pbyBuffer := ADR(ptSendData^[m_count]),(*geändert V1.4 bisher: [0] *)
								  diBufferSize := diSendCount-m_count,
								  diFlags :=m_Flags);
		CASE m_diReturn OF
		-1:	(* ERROR or data could not yet be send (V1.3 due to new FW11) *)
			m_ConnectionWatchdog(IN:=TRUE , PT:=tServerTimeOut );
			IF m_connectionWatchdog.Q THEN
				m_State:= STATE_CLOSE;
				m_ConnectionWatchdog(IN:=FALSE);(*reset connection watchdog*)
				diError := 16#8007;
			END_IF
		0: (* socket was "gracefully closed"  *)
			m_State := STATE_CLOSE;
			diError := 16#8003;
		ELSE (* succesful *)
			m_count:=m_count+m_diReturn;
			IF m_count>=diSendCount THEN
				diError := 16#0000;
				m_State := STATE_RX;
				m_count:=0;
				xStartSend:=FALSE;
			END_IF
			m_ConnectionWatchdog(IN:=FALSE);(*reset connection watchdog*)
		END_CASE


		STATE_CLOSE:	(* Close the server *)

		IF ADR(%MW0)=16#30000000  OR ADR(%MW0)=16#20000000 THEN (*841 or 881*)
			;
		ELSE
			IF m_Socket>=0 THEN
				SysSockShutdown(m_Socket, 0);;(*870*)
			END_IF
		END_IF
		IF m_Socket>=0 THEN
			SysSockClose( m_Socket);
		END_IF
		xClientConnected:= FALSE;
		m_State:= STATE_OPEN; (* Try to open the server again *)
		m_ConnectionWatchdog(IN:=FALSE);(*reset connection watchdog*)

		STATE_ERROR_TRAP: (* Error Read/Write socket  *)
			m_State:= STATE_ERROR_TRAP;

	ELSE  (* Bad FSM code trap  *)
			m_State:= STATE_ERROR_TRAP;
			diError:= 16#8008;
	END_CASE;
ELSE
	IF m_State <> STATE_INIT THEN
		IF ADR(%MW0)=16#30000000  OR ADR(%MW0)=16#20000000 THEN (*841 or 881*)
			;
		ELSE
			IF m_Socket>=0 THEN
				SysSockShutdown(m_Socket, 0);;(*870*)
			END_IF
		END_IF
		IF m_Socket>=0 THEN
			SysSockClose( m_Socket);
		END_IF
		IF ADR(%MW0)=16#30000000  OR ADR(%MW0)=16#20000000 THEN (*841 or 881*)
			;
		ELSE
			IF m_ServerSocket>=0 THEN
				SysSockShutdown(m_ServerSocket, 0);;(*870*)
			END_IF
		END_IF
		IF m_ServerSocket>=0 THEN
			SysSockClose( m_ServerSocket);
		END_IF
		xClientConnected:= FALSE;
		diError:= 0;
		m_State:= STATE_init; (* Try to open the server again *)
		m_ConnectionWatchdog(IN:=FALSE);(*reset connection watchdog*)
	END_IF
END_IF
END_FUNCTION_BLOCK

(* POU TCP_Logger/LogEv, ST *)
FUNCTION LogEv : BOOL
VAR_INPUT
	Level	: en_Logger_ErrLev;
	Object  : en_SYS_Objects;
	Index	: WORD;
	Error	: WORD;
	Message : STRING;
END_VAR
VAR
	s1 : STRING(160);
	i  : INT;
	Oggetto: STRING;
	NumeroOggetto: INT;
END_VAR
(* Execute error level operations *)

Sys.Alarm:=Lamp.SistemaInAllarme;
Sys.Warning:=Lamp.SistemaWarning;

NumeroOggetto:=Object;
CASE NumeroOggetto OF

	0: Oggetto:='SYS'; 					(* PLC *)
	1: Oggetto:='VPN' ;					(* VPN *)
	2: Oggetto:='DOOR' ;				(* Door & access control *)

	10: Oggetto:='CAL';				(* Caldaia *)
	11: Oggetto:='CIR' ;				(* Circolatore *)
	12: Oggetto:='CRON' ;				(* Crono-termostato *)
	13: Oggetto:='VRD' 	;				(* Valvola miscelatore pannelli *)
	14: Oggetto:='CTL'	;				(* Contalitri *)
	15: Oggetto:='CTB' 	;				(* Contabilizzatore *)
	16: Oggetto:='TPV' 	;				(* Temperature probes values *)
	17: Oggetto:='PPV' ;					(* Pressure probes values *)
	18: Oggetto:='PBV' 	;				(* Over-Pressure Alarms *)
	19: Oggetto:='TBV' 	;				(* Over-Temperature Alarms *)
	20: Oggetto:='PMV'	;				(* Under-Pressure Alarms *)
	21: Oggetto:='GRU'	;				(* Gruppo termico *)
	22:  Oggetto:='PDC' 	;				(* Pompa di calore *)
	23:  Oggetto:='SOL'	;				(* Pannello solare termico *)
	24:  Oggetto:='ESOL';				(* Pannello solare fotovoltaico *)
	25:  Oggetto:='GAS' ;			(* Contatore GAS *)
	26:  Oggetto:='PORT';				(* Misuratore di portata *)
	27:  Oggetto:='FPV' ;				(* Flow probes values *)
	28:  Oggetto:='ANZ' 	;				(* Analizzatore di rete *)
	29:  Oggetto:='SCA' 	;				(* Signal Control Alarms *)
	30:  Oggetto:='LUX' 	;				(* Base Illumination point *)
	31:  Oggetto:='LUXM';				(* Metered Illumination point *)
	32:  Oggetto:='PSG' ;				(* Sensore di passaggio *)
	33:  Oggetto:='HVAC' 	;			(* Heating, Ventilating and Air Conditioning *)
	34:  Oggetto:='HYGRV' 	;			(* Relative Humidity sensors value *)
	35:  Oggetto:='COOV'    ;			(* Carbon Dioxide CO2 sensors value *)
	36:  Oggetto:='INV'		;			(* Inverter *)
	37:  Oggetto:='STR'		;			(* Smart string box *)
	39:  Oggetto:='CIRD	' 	;			(* Double CIR *)
	40:  Oggetto:='ACS' 		;			(* Hot domestic water *)
	41:  Oggetto:='FRG' 		;			(* Frigo *)
	42:  Oggetto:='THER'	;			(* Thermostat *)
	43:  Oggetto:='CIRM	' ;				(* Modbus CIR *)
	44:  Oggetto:='CIRDM';				(* Modbus double CIR *)
	46:  Oggetto:='UTA' 	;				(* Modbus double CIR *)
	53:  Oggetto:='FPT'	;				(* Flow Pressure Temperature	FPTxx *)
	200:  Oggetto:='ZGW' ;				(* ZigBee - Gateway *)
	201:  Oggetto:='ZRM'	;			(* ZigBee - Repeater *)
	202:  Oggetto:='ZREL'	;			(* ZigBee - Actuator rele *)
	203:  Oggetto:='ZTHL';				(* ZigBee - Temperature Sensor *)
	250:  Oggetto:='ASGW'	;			(* ASi - Gateway *)
	251:  Oggetto:='ASCBI'	;			(* ASi - Input Board, Ciabatta *)
	1000:  Oggetto:='LON'	;			(* Bus - LON *)
	1001:  Oggetto:='MODBUS'; 			(* Bus - MODBUS *)
	1002:  Oggetto:='MBUS	' ;			(* Bus - M-BUS *)
	1003:  Oggetto:='MODBUS_TCP' ;	(* Bus - MODBUS TCP *)
	3000:  Oggetto:='VAR'; 				(* Variabili Generali di Set e Get *)
	10000:  Oggetto:='COMPINGRR'	;	(*Compressore Ingerson Rand R225 NE *)
	10001:  Oggetto:='COMPINGRML';	(*Compressore Ingerson Rand ML250SSR *)
	10002:  Oggetto:='ESC'	;			(*Essicatore *)

	9000:  Oggetto:='GENERIC'; 			(* Generic dataset *)
	9001:  Oggetto:='EXPO	';			(* EXPO dataset *)

ELSE
	Oggetto:='NonClasd';
END_CASE;

(* Aggiungo l'indice *)

		IF Index<10 THEN Oggetto:=CONCAT(Oggetto,'0');END_IF
		Oggetto:=CONCAT(Oggetto,WORD_TO_STRING(Index));









(* Fill lastlog list *)
s1:=CONCAT(Sys.Time_LogString,';Lev=');
s1:=CONCAT(s1,INT_TO_STRING(Level));
s1:=CONCAT(s1,';Obj=');
s1:=CONCAT(s1,INT_TO_STRING(Object));
s1:=CONCAT(s1,';Idx=');
s1:=CONCAT(s1,WORD_TO_STRING(Index));
s1:=CONCAT(s1,';Err=');
s1:=CONCAT(s1,WORD_TO_STRING(Error));
s1:=CONCAT(s1,';');
s1:=CONCAT(s1,Oggetto);


Sys.LastLogs_Dat[Sys.LastLogs_Idx]:=s1;
Sys.LastLogs_Msg[Sys.LastLogs_Idx]:=Message;
Sys.LastLogs_Idx:=Sys.LastLogs_Idx+1;
IF Sys.LastLogs_Idx>5 THEN Sys.LastLogs_Idx:=0; END_IF

(*---------------------------------------------------------------*)
	Logger_Head();
(*---------------------------------------------------------------*)

(* Insert ERR *)
s1:=CONCAT('&ERR=',INT_TO_STRING(Level));
s1:=CONCAT(s1,';');
s1:=CONCAT(s1,INT_TO_STRING(Object));
s1:=CONCAT(s1,';');
s1:=CONCAT(s1,WORD_TO_STRING(Index));
s1:=CONCAT(s1,';');
s1:=CONCAT(s1,WORD_TO_STRING(Error));
s1:=CONCAT(s1,';');
ADDSTRING(ADR(Logger.TData), ADR(s1), Logger.TLen);
s1:=Message;
STR_NOSPACES(ADR(s1));
ADDSTRING(ADR(Logger.TData), ADR(s1), Logger.TLen);
s1:=CONCAT(s1,';');
s1:=CONCAT(s1,Oggetto);
STR_NOSPACES(ADR(s1));
ADDSTRING(ADR(Logger.TData), ADR(s1), Logger.TLen);

(*---------------------------------------------------------------*)
	Logger_Send();
(*---------------------------------------------------------------*)
END_FUNCTION

(* POU TCP_Logger/Logger_Head, ST *)
FUNCTION Logger_Head : BOOL
VAR
	s1 : STRING(160);
	i  : BYTE;
END_VAR
Logger.TLen:=0;
(* Set GET header *)
ADDSTRING(ADR(Logger.TData), ADR(Logger_GETSTART), Logger.TLen);

(* Insert Header *)
s1:=INSERT('ID=&V=1&D=',DWORD_TO_STRING(Plant_SN),3);
s1:=CONCAT(s1,REPLACE(Sys.Time_LogString,'T',1,11));
(*s1:=CONCAT(s1,Sys.Time_LogString) *)
s1:=CONCAT(s1,'&S=');
IF Sys.Alarm THEN i:=2; ELSIF Sys.Warning THEN i:=1; ELSE i:=0; END_IF
s1:=CONCAT(s1,BYTE_TO_STRING(i));
ADDSTRING(ADR(Logger.TData), ADR(s1), Logger.TLen);
END_FUNCTION

(* POU Utils Functions/ADDSTRING, ST *)
FUNCTION ADDSTRING : BOOL
VAR_INPUT
	pTxData: POINTER TO BYTE;
	pString: POINTER TO BYTE;
END_VAR
VAR_IN_OUT
	TxLen: DINT;
END_VAR
VAR
END_VAR
pTxData:=pTxData+TxLen;
WHILE pString^<>0 DO
	pTxData^:=pString^;
	pString:=pString+1;
	pTxData:=pTxData+1;
	TxLen:=TxLen+1;
END_WHILE
END_FUNCTION

(* POU Utils Functions/STR_NOSPACES, ST *)
FUNCTION STR_NOSPACES : BOOL (* Replace spaces and bad chars with allowed ones, used as HTTP-GET validator *)
VAR_INPUT
	pString: POINTER TO BYTE;
END_VAR
VAR
END_VAR
WHILE pString^<>0 DO
	IF pString^=16#20 (* space *) THEN pString^:=16#5F; (*'_'*) END_IF
	pString:=pString+1;
END_WHILE
END_FUNCTION

(* POU TCP_Logger/Logger_Send, ST *)
FUNCTION Logger_Send : BOOL
VAR
	hFile: 	DWORD;
	pos:	DWORD;
	myDataFileOLD:STRING(255);

END_VAR
(* Finalize string *)
ADDSTRING(ADR(Logger.TData), ADR(Logger_GETEND), Logger.TLen);

(* Read log position *)
pos:=SysFileGetSize(Logger_DataFile);
(* Check log size, bckup and erase if no pending messages *)
IF pos>5000000(*5M*) THEN
	hFile:=SysFileOpen(Logger_IndexFile,'r');
	IF hFile=0 THEN

		(*backup management with multiple files*)
		IF LogBCKIndex>0 AND LogBCKIndex <Logger_MaxBCK THEN
			LogBCKIndex:=LogBCKIndex+1;
		ELSE
			LogBCKIndex:=1;
		END_IF

		myDataFileOLD:=CONCAT(Logger_DataFileOld,WORD_TO_STRING(LogBCKIndex));
		SysFileDelete(myDataFileOLD);
		SysFileRename(Logger_DataFile,myDataFileOLD);
		pos:=0;
	ELSE
		SysFileClose(hFile);
	END_IF
END_IF
(* Write message on log file *)
hFile:=SysFileOpen(Logger_DataFile,'a');
IF hFile<>0 THEN
	SysFileWrite(hFile, ADR(Logger.TData), Logger.TLen);
	SysFileClose(hFile);
ELSE
	Sys.Warning:=TRUE;
END_IF


(* Check logger status *)
IF Logger.SendReq=FALSE THEN
	(* Set log position for recovery *)
	Logger.SendIdx:=pos;
	(* Copy message data *)
	MEMCPY(ADR(Logger.TData),ADR(Logger.SendData),DINT_TO_WORD(Logger.TLen));
	Logger.SendLen:=Logger.TLen;
	(* Trigger request *)
	Logger.SendReq:=TRUE;
ELSE
	(* Add message position+size in recovery indexes *)
	hFile:=SysFileOpen(Logger_IndexFile,'a');
	SysFileWrite(hFile, ADR(pos), SIZEOF(pos));
	SysFileWrite(hFile, ADR(Logger.TLen), SIZEOF(Logger.TLen));
	SysFileClose(hFile);
END_IF
END_FUNCTION

(* POU Utils Functions/MEMCPY, ST *)
FUNCTION MEMCPY:BOOL
VAR_INPUT
	pSourceAddress:POINTER TO ARRAY[1..2] OF BYTE;
	pDestinationAddress:POINTER TO ARRAY[1..2] OF BYTE;
	BytesToCopy:WORD;
END_VAR
VAR
END_VAR
WHILE (BytesToCopy > 0) DO
	pDestinationAddress^[1]:=pSourceAddress^[1]; (* copy bytes from source to destination *)
	pDestinationAddress:=ADR(pDestinationAddress^[2]); (* increment destination *)
	pSourceAddress:=ADR(pSourceAddress^[2]);(* increment source *)
	BytesToCopy:=BytesToCopy -1; (* decrement number of bytes to copy *)
END_WHILE
END_FUNCTION

